# B&R Automation Studio project mvDemoTrak
Automation Studio 4.12.3.127 SP; technology packages: mapp 5.22.1, mappCockpit 5.22.0, mappMotion 5.22.1, mappView 5.22.1

## Configuration CP1685

CPU X20CP1685, AutomationRuntime D4.93, Build 6.3.0, Safety 0.0, Vc 

### Task classes (Cpu.sw)
```
Cyclic#1 (cycle 2000 us, tolerance 0 us):
  VisuTask <- VisuPackage.VisuTask.prg
Cyclic#2 (cycle 10000 us, tolerance 10000 us):
  AlarmXTask <- VisuPackage.AlarmXTask.prg
Binaries: FWRules, arsvcreg, TCData, TCLang, udbdef, mvLoader, CfgAlList, iomap, TC, Role, arconfig, asfw, ashwac, sysconf, CfgAlHist, User, ashwd
Libraries: standard, MpAlarmX, MpBase, astime, runtime, MpServer, AsBrStr, sys_lib, asieccon, arssl, dataobj, aruser, McBase, CoTrace, AsZip, FileIO
```

### Hardware
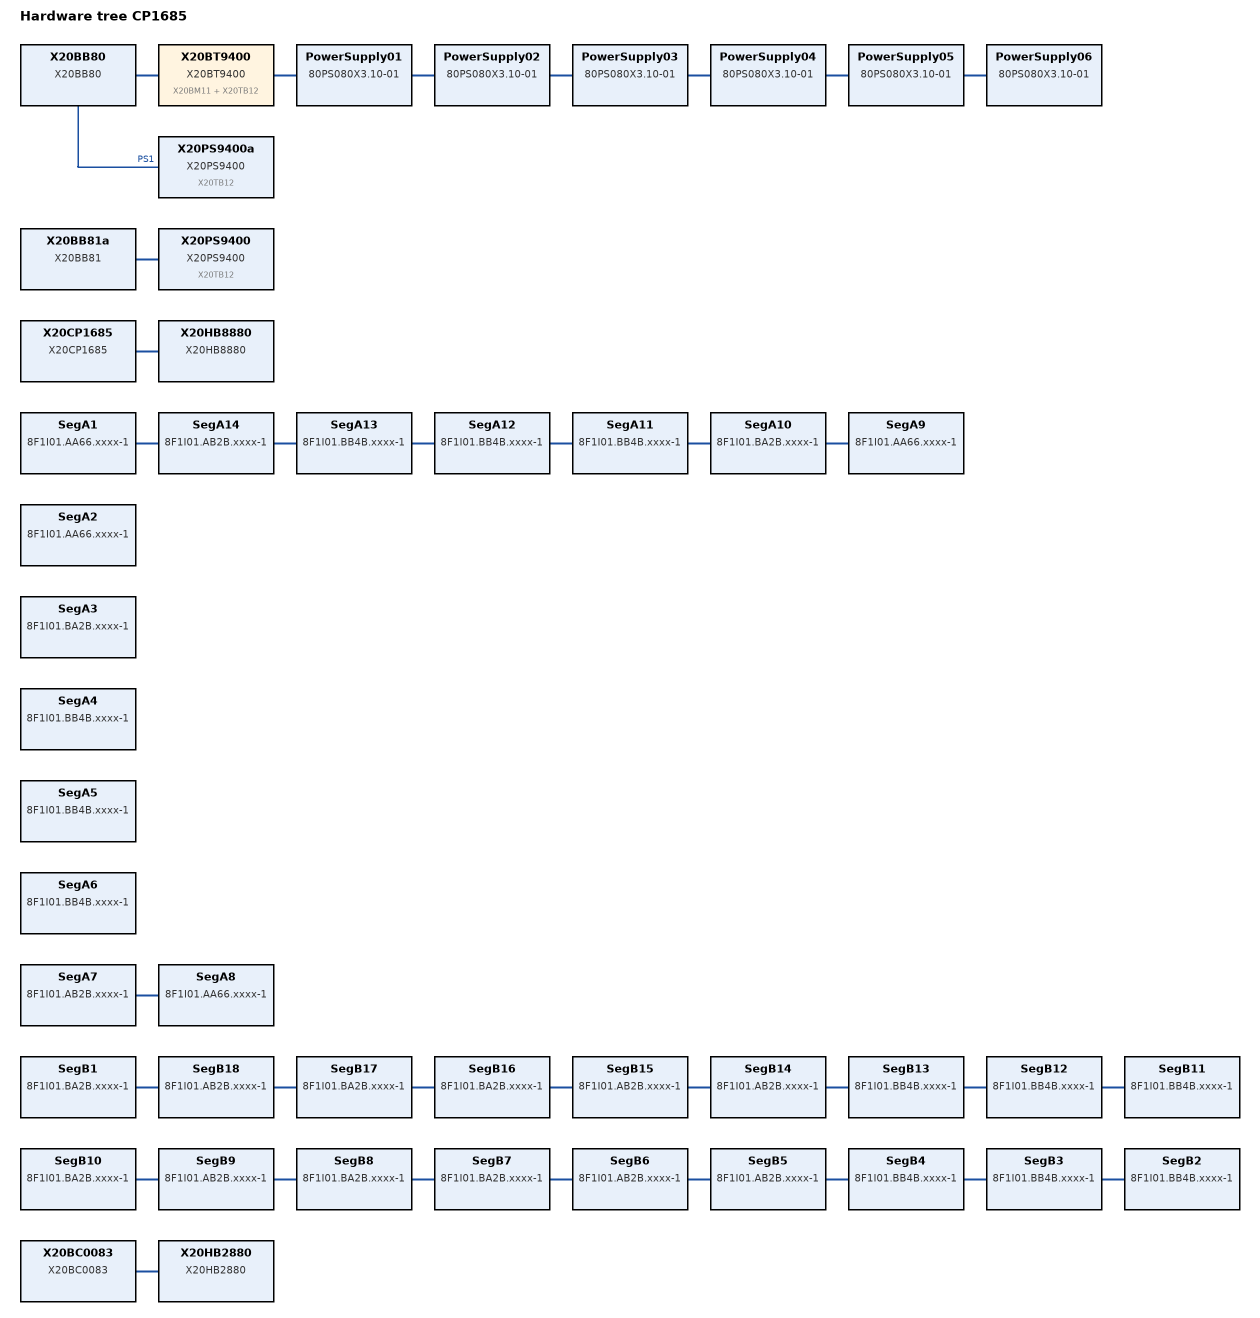
```
PowerSupply01 : 80PS080X3.10-01 v1.5.0.0  [X2X1 -> X20BT9400.X2X1 [Cable Type=X2XCable, Length=10, Version=1.0.0.3]]
  Supervision = off
PowerSupply02 : 80PS080X3.10-01 v1.5.0.0  [X2X1 -> PowerSupply01.X2X2 [Cable Type=X2XCable, Length=10, Version=1.0.0.3]]
  Supervision = off
PowerSupply03 : 80PS080X3.10-01 v1.5.0.0  [X2X1 -> PowerSupply02.X2X2 [Cable Type=X2XCable, Length=10, Version=1.0.0.3]]
  Supervision = off
PowerSupply04 : 80PS080X3.10-01 v1.5.0.0  [X2X1 -> PowerSupply03.X2X2 [Cable Type=X2XCable, Length=10, Version=1.0.0.3]]
  Supervision = off
PowerSupply05 : 80PS080X3.10-01 v1.5.0.0  [X2X1 -> PowerSupply04.X2X2 [Cable Type=X2XCable, Length=10, Version=1.0.0.3]]
  Supervision = off
PowerSupply06 : 80PS080X3.10-01 v1.5.0.0  [X2X1 -> PowerSupply05.X2X2 [Cable Type=X2XCable, Length=10, Version=1.0.0.3]]
  Supervision = off
SegA1 : 8F1I01.AA66.xxxx-1 v1.0.0.2  [PLK1 -> SegA2.PLK2 (NodeNumber=1) [Cable Type=PowerlinkCable, Length=10, Version=1.0.0.3]; PLK2 -> SegA14.PLK1 (NodeNumber=1) [Cable Type=PowerlinkCable, Length=10, Version=1.0.0.3]; PLK3 -> X20HB8880.ETH2 (NodeNumber=1) [Cable Type=PowerlinkCable, Length=10, Version=1.0.0.3]]
  DriveConfiguration:
    McTypeID = LLMConfig
  DriveConfiguration/Segment:
    Shape = STRAIGHT660
    SegmentReference = gSegA1
    SegmentSectorDirection = Positive
    ElongationCompensation = UseAssemblySetting
    StopReaction = UseAssemblySetting
    SpeedFilter = UseAssemblySetting
SegA10 : 8F1I01.BA2B.xxxx-1 v1.0.0.2  [PLK1 -> SegA11.PLK2 (NodeNumber=25) [Cable Type=PowerlinkCable, Length=10, Version=1.0.0.3]; PLK2 -> SegA9.PLK1 (NodeNumber=25) [Cable Type=PowerlinkCable, Length=10, Version=1.0.0.3]]
  DriveConfiguration:
    McTypeID = LLMConfig
  DriveConfiguration/Segment:
    Shape = CIRCULAR_TO_STRAIGHT105
    SegmentReference = gSegA10
    SegmentSectorDirection = Positive
    ElongationCompensation = UseAssemblySetting
    StopReaction = UseAssemblySetting
    SpeedFilter = UseAssemblySetting
SegA11 : 8F1I01.BB4B.xxxx-1 v1.0.0.2  [PLK1 -> SegA12.PLK2 (NodeNumber=24) [Cable Type=PowerlinkCable, Length=10, Version=1.0.0.3]; PLK2 -> SegA10.PLK1 (NodeNumber=24) [Cable Type=PowerlinkCable, Length=10, Version=1.0.0.3]]
  DriveConfiguration:
    McTypeID = LLMConfig
  DriveConfiguration/Segment:
    Shape = CIRCULAR
    SegmentReference = gSegA11
    SegmentSectorDirection = Positive
    ElongationCompensation = UseAssemblySetting
    StopReaction = UseAssemblySetting
    SpeedFilter = UseAssemblySetting
SegA12 : 8F1I01.BB4B.xxxx-1 v1.0.0.2  [PLK1 -> SegA13.PLK2 (NodeNumber=23) [Cable Type=PowerlinkCable, Length=10, Version=1.0.0.3]; PLK2 -> SegA11.PLK1 (NodeNumber=23) [Cable Type=PowerlinkCable, Length=10, Version=1.0.0.3]]
  DriveConfiguration:
    McTypeID = LLMConfig
  DriveConfiguration/Segment:
    Shape = CIRCULAR
    SegmentReference = gSegA12
    SegmentSectorDirection = Positive
    ElongationCompensation = UseAssemblySetting
    StopReaction = UseAssemblySetting
    SpeedFilter = UseAssemblySetting
SegA13 : 8F1I01.BB4B.xxxx-1 v1.0.0.2  [PLK1 -> SegA14.PLK2 (NodeNumber=22) [Cable Type=PowerlinkCable, Length=10, Version=1.0.0.3]; PLK2 -> SegA12.PLK1 (NodeNumber=22) [Cable Type=PowerlinkCable, Length=10, Version=1.0.0.3]]
  DriveConfiguration:
    McTypeID = LLMConfig
  DriveConfiguration/Segment:
    Shape = CIRCULAR
    SegmentReference = gSegA13
    SegmentSectorDirection = Positive
    ElongationCompensation = UseAssemblySetting
    StopReaction = UseAssemblySetting
    SpeedFilter = UseAssemblySetting
SegA14 : 8F1I01.AB2B.xxxx-1 v1.0.0.2  [PLK1 -> SegA1.PLK2 (NodeNumber=21) [Cable Type=PowerlinkCable, Length=10, Version=1.0.0.3]; PLK2 -> SegA13.PLK1 (NodeNumber=21) [Cable Type=PowerlinkCable, Length=10, Version=1.0.0.3]]
  DriveConfiguration:
    McTypeID = LLMConfig
  DriveConfiguration/Segment:
    Shape = STRAIGHT105_TO_CIRCULAR
    SegmentReference = gSegA14
    SegmentSectorDirection = Positive
    ElongationCompensation = UseAssemblySetting
    StopReaction = UseAssemblySetting
    SpeedFilter = UseAssemblySetting
SegA2 : 8F1I01.AA66.xxxx-1 v1.0.0.2  [PLK1 -> SegA3.PLK2 (NodeNumber=2) [Cable Type=PowerlinkCable, Length=10, Version=1.0.0.3]; PLK2 -> SegA1.PLK1 (NodeNumber=2) [Cable Type=PowerlinkCable, Length=10, Version=1.0.0.3]]
  DriveConfiguration:
    McTypeID = LLMConfig
  DriveConfiguration/Segment:
    Shape = STRAIGHT660
    SegmentReference = gSegA2
    SegmentSectorDirection = Positive
    ElongationCompensation = UseAssemblySetting
    StopReaction = UseAssemblySetting
    SpeedFilter = UseAssemblySetting
SegA3 : 8F1I01.BA2B.xxxx-1 v1.0.0.2  [PLK1 -> SegA4.PLK2 (NodeNumber=27) [Cable Type=PowerlinkCable, Length=10, Version=1.0.0.3]; PLK2 -> SegA2.PLK1 (NodeNumber=27) [Cable Type=PowerlinkCable, Length=10, Version=1.0.0.3]]
  DriveConfiguration:
    McTypeID = LLMConfig
  DriveConfiguration/Segment:
    Shape = CIRCULAR_TO_STRAIGHT105
    SegmentReference = gSegA3
    SegmentSectorDirection = Positive
    ElongationCompensation = UseAssemblySetting
    StopReaction = UseAssemblySetting
    SpeedFilter = UseAssemblySetting
SegA4 : 8F1I01.BB4B.xxxx-1 v1.0.0.2  [PLK1 -> SegA5.PLK2 (NodeNumber=28) [Cable Type=PowerlinkCable, Length=10, Version=1.0.0.3]; PLK2 -> SegA3.PLK1 (NodeNumber=28) [Cable Type=PowerlinkCable, Length=10, Version=1.0.0.3]]
  DriveConfiguration:
    McTypeID = LLMConfig
  DriveConfiguration/Segment:
    Shape = CIRCULAR
    SegmentReference = gSegA4
    SegmentSectorDirection = Positive
    ElongationCompensation = UseAssemblySetting
    StopReaction = UseAssemblySetting
    SpeedFilter = UseAssemblySetting
SegA5 : 8F1I01.BB4B.xxxx-1 v1.0.0.2  [PLK1 -> SegA6.PLK2 (NodeNumber=29) [Cable Type=PowerlinkCable, Length=10, Version=1.0.0.3]; PLK2 -> SegA4.PLK1 (NodeNumber=29) [Cable Type=PowerlinkCable, Length=10, Version=1.0.0.3]]
  DriveConfiguration:
    McTypeID = LLMConfig
  DriveConfiguration/Segment:
    Shape = CIRCULAR
    SegmentReference = gSegA5
    SegmentSectorDirection = Positive
    ElongationCompensation = UseAssemblySetting
    StopReaction = UseAssemblySetting
    SpeedFilter = UseAssemblySetting
SegA6 : 8F1I01.BB4B.xxxx-1 v1.0.0.2  [PLK1 -> SegA7.PLK2 (NodeNumber=30) [Cable Type=PowerlinkCable, Length=10, Version=1.0.0.3]; PLK2 -> SegA5.PLK1 (NodeNumber=30) [Cable Type=PowerlinkCable, Length=10, Version=1.0.0.3]]
  DriveConfiguration:
    McTypeID = LLMConfig
  DriveConfiguration/Segment:
    Shape = CIRCULAR
    SegmentReference = gSegA6
    SegmentSectorDirection = Positive
    ElongationCompensation = UseAssemblySetting
    StopReaction = UseAssemblySetting
    SpeedFilter = UseAssemblySetting
SegA7 : 8F1I01.AB2B.xxxx-1 v1.0.0.2  [PLK1 -> SegA8.PLK2 (NodeNumber=31) [Cable Type=PowerlinkCable, Length=10, Version=1.0.0.3]; PLK2 -> SegA6.PLK1 (NodeNumber=31) [Cable Type=PowerlinkCable, Length=10, Version=1.0.0.3]]
  DriveConfiguration:
    McTypeID = LLMConfig
  DriveConfiguration/Segment:
    Shape = STRAIGHT105_TO_CIRCULAR
    SegmentReference = gSegA7
    SegmentSectorDirection = Positive
    ElongationCompensation = UseAssemblySetting
    StopReaction = UseAssemblySetting
    SpeedFilter = UseAssemblySetting
SegA8 : 8F1I01.AA66.xxxx-1 v1.0.0.2  [PLK2 -> SegA7.PLK1 (NodeNumber=32) [Cable Type=PowerlinkCable, Length=10, Version=1.0.0.3]]
  DriveConfiguration:
    McTypeID = LLMConfig
  DriveConfiguration/Segment:
    Shape = STRAIGHT660
    SegmentReference = gSegA8
    SegmentSectorDirection = Positive
    ElongationCompensation = UseAssemblySetting
    StopReaction = UseAssemblySetting
    SpeedFilter = UseAssemblySetting
SegA9 : 8F1I01.AA66.xxxx-1 v1.0.0.2  [PLK1 -> SegA10.PLK2 (NodeNumber=26) [Cable Type=PowerlinkCable, Length=10, Version=1.0.0.3]]
  DriveConfiguration:
    McTypeID = LLMConfig
  DriveConfiguration/Segment:
    Shape = STRAIGHT660
    SegmentReference = gSegA9
    SegmentSectorDirection = Positive
    ElongationCompensation = UseAssemblySetting
    StopReaction = UseAssemblySetting
    SpeedFilter = UseAssemblySetting
SegB1 : 8F1I01.BA2B.xxxx-1 v1.0.0.2  [PLK1 -> SegB2.PLK2 (NodeNumber=3) [Cable Type=PowerlinkCable, Length=10, Version=1.0.0.3]; PLK2 -> SegB18.PLK1 (NodeNumber=3) [Cable Type=PowerlinkCable, Length=10, Version=1.0.0.3]; PLK3 -> X20HB2880.ETH2 (NodeNumber=3) [Cable Type=PowerlinkCable, Length=10, Version=1.0.0.3]]
  DriveConfiguration:
    McTypeID = LLMConfig
  DriveConfiguration/Segment:
    Shape = CIRCULAR_TO_STRAIGHT105
    SegmentReference = gSegB1
    SegmentSectorDirection = Positive
    ElongationCompensation = UseAssemblySetting
    StopReaction = UseAssemblySetting
    SpeedFilter = UseAssemblySetting
SegB10 : 8F1I01.BA2B.xxxx-1 v1.0.0.2  [PLK2 -> SegB9.PLK1 (NodeNumber=12) [Cable Type=PowerlinkCable, Length=10, Version=1.0.0.3]]
  DriveConfiguration:
    McTypeID = LLMConfig
  DriveConfiguration/Segment:
    Shape = CIRCULAR_TO_STRAIGHT105
    SegmentReference = gSegB10
    SegmentSectorDirection = Positive
    ElongationCompensation = UseAssemblySetting
    StopReaction = UseAssemblySetting
    SpeedFilter = UseAssemblySetting
SegB11 : 8F1I01.BB4B.xxxx-1 v1.0.0.2  [PLK1 -> SegB12.PLK2 (NodeNumber=11) [Cable Type=PowerlinkCable, Length=10, Version=1.0.0.3]]
  DriveConfiguration:
    McTypeID = LLMConfig
  DriveConfiguration/Segment:
    Shape = CIRCULAR
    SegmentReference = gSegB11
    SegmentSectorDirection = Positive
    ElongationCompensation = UseAssemblySetting
    StopReaction = UseAssemblySetting
    SpeedFilter = UseAssemblySetting
SegB12 : 8F1I01.BB4B.xxxx-1 v1.0.0.2  [PLK1 -> SegB13.PLK2 (NodeNumber=10) [Cable Type=PowerlinkCable, Length=10, Version=1.0.0.3]; PLK2 -> SegB11.PLK1 (NodeNumber=10) [Cable Type=PowerlinkCable, Length=10, Version=1.0.0.3]]
  DriveConfiguration:
    McTypeID = LLMConfig
  DriveConfiguration/Segment:
    Shape = CIRCULAR
    SegmentReference = gSegB12
    SegmentSectorDirection = Positive
    ElongationCompensation = UseAssemblySetting
    StopReaction = UseAssemblySetting
    SpeedFilter = UseAssemblySetting
SegB13 : 8F1I01.BB4B.xxxx-1 v1.0.0.2  [PLK1 -> SegB14.PLK2 (NodeNumber=9) [Cable Type=PowerlinkCable, Length=10, Version=1.0.0.3]; PLK2 -> SegB12.PLK1 (NodeNumber=9) [Cable Type=PowerlinkCable, Length=10, Version=1.0.0.3]]
  DriveConfiguration:
    McTypeID = LLMConfig
  DriveConfiguration/Segment:
    Shape = CIRCULAR
    SegmentReference = gSegB13
    SegmentSectorDirection = Positive
    ElongationCompensation = UseAssemblySetting
    StopReaction = UseAssemblySetting
    SpeedFilter = UseAssemblySetting
SegB14 : 8F1I01.AB2B.xxxx-1 v1.0.0.2  [PLK1 -> SegB15.PLK2 (NodeNumber=8) [Cable Type=PowerlinkCable, Length=10, Version=1.0.0.3]; PLK2 -> SegB13.PLK1 (NodeNumber=8) [Cable Type=PowerlinkCable, Length=10, Version=1.0.0.3]]
  DriveConfiguration:
    McTypeID = LLMConfig
  DriveConfiguration/Segment:
    Shape = STRAIGHT105_TO_CIRCULAR
    SegmentReference = gSegB14
    SegmentSectorDirection = Positive
    ElongationCompensation = UseAssemblySetting
    StopReaction = UseAssemblySetting
    SpeedFilter = UseAssemblySetting
SegB15 : 8F1I01.AB2B.xxxx-1 v1.0.0.2  [PLK1 -> SegB16.PLK2 (NodeNumber=7) [Cable Type=PowerlinkCable, Length=10, Version=1.0.0.3]; PLK2 -> SegB14.PLK1 (NodeNumber=7) [Cable Type=PowerlinkCable, Length=10, Version=1.0.0.3]]
  DriveConfiguration:
    McTypeID = LLMConfig
  DriveConfiguration/Segment:
    Shape = STRAIGHT105_TO_CIRCULAR
    SegmentReference = gSegB15
    SegmentSectorDirection = Positive
    ElongationCompensation = UseAssemblySetting
    StopReaction = UseAssemblySetting
    SpeedFilter = UseAssemblySetting
SegB16 : 8F1I01.BA2B.xxxx-1 v1.0.0.2  [PLK1 -> SegB17.PLK2 (NodeNumber=6) [Cable Type=PowerlinkCable, Length=10, Version=1.0.0.3]; PLK2 -> SegB15.PLK1 (NodeNumber=6) [Cable Type=PowerlinkCable, Length=10, Version=1.0.0.3]]
  DriveConfiguration:
    McTypeID = LLMConfig
  DriveConfiguration/Segment:
    Shape = CIRCULAR_TO_STRAIGHT105
    SegmentReference = gSegB16
    SegmentSectorDirection = Positive
    ElongationCompensation = UseAssemblySetting
    StopReaction = UseAssemblySetting
    SpeedFilter = UseAssemblySetting
SegB17 : 8F1I01.BA2B.xxxx-1 v1.0.0.2  [PLK1 -> SegB18.PLK2 (NodeNumber=5) [Cable Type=PowerlinkCable, Length=10, Version=1.0.0.3]; PLK2 -> SegB16.PLK1 (NodeNumber=5) [Cable Type=PowerlinkCable, Length=10, Version=1.0.0.3]]
  DriveConfiguration:
    McTypeID = LLMConfig
  DriveConfiguration/Segment:
    Shape = CIRCULAR_TO_STRAIGHT105
    SegmentReference = gSegB17
    SegmentSectorDirection = Positive
    ElongationCompensation = UseAssemblySetting
    StopReaction = UseAssemblySetting
    SpeedFilter = UseAssemblySetting
SegB18 : 8F1I01.AB2B.xxxx-1 v1.0.0.2  [PLK1 -> SegB1.PLK2 (NodeNumber=4) [Cable Type=PowerlinkCable, Length=10, Version=1.0.0.3]; PLK2 -> SegB17.PLK1 (NodeNumber=4) [Cable Type=PowerlinkCable, Length=10, Version=1.0.0.3]]
  DriveConfiguration:
    McTypeID = LLMConfig
  DriveConfiguration/Segment:
    Shape = STRAIGHT105_TO_CIRCULAR
    SegmentReference = gSegB18
    SegmentSectorDirection = Positive
    ElongationCompensation = UseAssemblySetting
    StopReaction = UseAssemblySetting
    SpeedFilter = UseAssemblySetting
SegB2 : 8F1I01.BB4B.xxxx-1 v1.0.0.2  [PLK1 -> SegB3.PLK2 (NodeNumber=13) [Cable Type=PowerlinkCable, Length=10, Version=1.0.0.3]; PLK2 -> SegB1.PLK1 (NodeNumber=13) [Cable Type=PowerlinkCable, Length=10, Version=1.0.0.3]]
  DriveConfiguration:
    McTypeID = LLMConfig
  DriveConfiguration/Segment:
    Shape = CIRCULAR
    SegmentReference = gSegB2
    SegmentSectorDirection = Positive
    ElongationCompensation = UseAssemblySetting
    StopReaction = UseAssemblySetting
    SpeedFilter = UseAssemblySetting
SegB3 : 8F1I01.BB4B.xxxx-1 v1.0.0.2  [PLK1 -> SegB4.PLK2 (NodeNumber=14) [Cable Type=PowerlinkCable, Length=10, Version=1.0.0.3]; PLK2 -> SegB2.PLK1 (NodeNumber=14) [Cable Type=PowerlinkCable, Length=10, Version=1.0.0.3]]
  DriveConfiguration:
    McTypeID = LLMConfig
  DriveConfiguration/Segment:
    Shape = CIRCULAR
    SegmentReference = gSegB3
    SegmentSectorDirection = Positive
    ElongationCompensation = UseAssemblySetting
    StopReaction = UseAssemblySetting
    SpeedFilter = UseAssemblySetting
SegB4 : 8F1I01.BB4B.xxxx-1 v1.0.0.2  [PLK1 -> SegB5.PLK2 (NodeNumber=15) [Cable Type=PowerlinkCable, Length=10, Version=1.0.0.3]; PLK2 -> SegB3.PLK1 (NodeNumber=15) [Cable Type=PowerlinkCable, Length=10, Version=1.0.0.3]]
  DriveConfiguration:
    McTypeID = LLMConfig
  DriveConfiguration/Segment:
    Shape = CIRCULAR
    SegmentReference = gSegB4
    SegmentSectorDirection = Positive
    ElongationCompensation = UseAssemblySetting
    StopReaction = UseAssemblySetting
    SpeedFilter = UseAssemblySetting
SegB5 : 8F1I01.AB2B.xxxx-1 v1.0.0.2  [PLK1 -> SegB6.PLK2 (NodeNumber=16) [Cable Type=PowerlinkCable, Length=10, Version=1.0.0.3]; PLK2 -> SegB4.PLK1 (NodeNumber=16) [Cable Type=PowerlinkCable, Length=10, Version=1.0.0.3]]
  DriveConfiguration:
    McTypeID = LLMConfig
  DriveConfiguration/Segment:
    Shape = STRAIGHT105_TO_CIRCULAR
    SegmentReference = gSegB5
    SegmentSectorDirection = Positive
    ElongationCompensation = UseAssemblySetting
    StopReaction = UseAssemblySetting
    SpeedFilter = UseAssemblySetting
SegB6 : 8F1I01.AB2B.xxxx-1 v1.0.0.2  [PLK1 -> SegB7.PLK2 (NodeNumber=17) [Cable Type=PowerlinkCable, Length=10, Version=1.0.0.3]; PLK2 -> SegB5.PLK1 (NodeNumber=17) [Cable Type=PowerlinkCable, Length=10, Version=1.0.0.3]]
  DriveConfiguration:
    McTypeID = LLMConfig
  DriveConfiguration/Segment:
    Shape = STRAIGHT105_TO_CIRCULAR
    SegmentReference = gSegB6
    SegmentSectorDirection = Positive
    ElongationCompensation = UseAssemblySetting
    StopReaction = UseAssemblySetting
    SpeedFilter = UseAssemblySetting
SegB7 : 8F1I01.BA2B.xxxx-1 v1.0.0.2  [PLK1 -> SegB8.PLK2 (NodeNumber=18) [Cable Type=PowerlinkCable, Length=10, Version=1.0.0.3]; PLK2 -> SegB6.PLK1 (NodeNumber=18) [Cable Type=PowerlinkCable, Length=10, Version=1.0.0.3]]
  DriveConfiguration:
    McTypeID = LLMConfig
  DriveConfiguration/Segment:
    Shape = CIRCULAR_TO_STRAIGHT105
    SegmentReference = gSegB7
    SegmentSectorDirection = Positive
    ElongationCompensation = UseAssemblySetting
    StopReaction = UseAssemblySetting
    SpeedFilter = UseAssemblySetting
SegB8 : 8F1I01.BA2B.xxxx-1 v1.0.0.2  [PLK1 -> SegB9.PLK2 (NodeNumber=20) [Cable Type=PowerlinkCable, Length=10, Version=1.0.0.3]; PLK2 -> SegB7.PLK1 (NodeNumber=20) [Cable Type=PowerlinkCable, Length=10, Version=1.0.0.3]]
  DriveConfiguration:
    McTypeID = LLMConfig
  DriveConfiguration/Segment:
    Shape = CIRCULAR_TO_STRAIGHT105
    SegmentReference = gSegB8
    SegmentSectorDirection = Positive
    ElongationCompensation = UseAssemblySetting
    StopReaction = UseAssemblySetting
    SpeedFilter = UseAssemblySetting
SegB9 : 8F1I01.AB2B.xxxx-1 v1.0.0.2  [PLK1 -> SegB10.PLK2 (NodeNumber=19) [Cable Type=PowerlinkCable, Length=10, Version=1.0.0.3]; PLK2 -> SegB8.PLK1 (NodeNumber=19) [Cable Type=PowerlinkCable, Length=10, Version=1.0.0.3]]
  DriveConfiguration:
    McTypeID = LLMConfig
  DriveConfiguration/Segment:
    Shape = STRAIGHT105_TO_CIRCULAR
    SegmentReference = gSegB9
    SegmentSectorDirection = Positive
    ElongationCompensation = UseAssemblySetting
    StopReaction = UseAssemblySetting
    SpeedFilter = UseAssemblySetting
X20BB80 : X20BB80 v1.1.0.0
X20BB81a : X20BB81 v1.1.0.0
  Connector IF1:
    ActivateX2X = 0
X20BC0083 : X20BC0083 v2.14.0.0  [PLK1 -> X20HB2880.ETH1 (NodeNumber=33) [Cable Type=PowerlinkCable, Length=10, Version=1.0.0.3]; SL -> X20BB80.SL1]
  Supervision = off
X20BM11 : X20BM11 v1.1.0.0  [X2X1 -> X20BB80.IF1]
X20BT9400 : X20BT9400 v1.3.0.0  [SS1 -> X20TB12b.SS; SL -> X20BM11.SL1]
  Supervision = off
X20CP1685 : X20CP1685 v1.7.2.0
  Connector IF2:
    ActivateDevice = 1
    Mode = Manual
    InternetAddress = 192.168.0.105  // //10.49.40.211
    SubnetMask = 255.255.255.0
    ActivateSnmp = 2
  ConfigurationID = mvDemoTrak_CP1685
  MotionLoggerSize = 2048000
  EnableUsbRemoteInstall = 1
  TimerDeviceType = EPLX2X
  TimerDevice = X20CP1685.IF3
  TaskClassIdleTime = 2000
  Cyclic1Duration = 2000
  Cyclic1Tolerance = 0
  Cyclic2Duration = 10000
  Cyclic2Tolerance = 10000
  FileDevice1
  FileDeviceName1 = SvgData
  FileDevicePath1 = F:\web\SvgData
  FileDevice2
  FileDeviceName2 = Diagnosis
  FileDevicePath2 = F:\web\Diagnosis
  FtpUser1
  FtpUsername1 = Admin
  FtpUserPassword1 = b2dkeklN0DR4HlzomfG8N5dlVtI3Hrgd5HBjTL6T4A4=  // pw: admin
  FtpUserSalt1 = LZ6GLOae
  FTPAccessRight1 = 0
  FTPdevice1 = ALL
  WebServerWebDir = F:\web  // default: web\
  ActivateOpcUa = 1
  OpcUaInformationModels_PV_Version = 1
X20HB2880 : X20HB2880 v1.2.0.0  [ETH1 -> X20BC0083.PLK1 [Cable Type=PowerlinkCable, Length=10, Version=1.0.0.3]; ETH2 -> SegB1.PLK3 [Cable Type=PowerlinkCable, Length=10, Version=1.0.0.3]; SS -> X20BB81a.SS1]
X20HB8880 : X20HB8880 v1.1.0.0  [ETH1 -> X20CP1685.IF3 [Cable Type=PowerlinkCable, Length=10, Version=1.0.0.3]; ETH2 -> SegA1.PLK3 [Cable Type=PowerlinkCable, Length=10, Version=1.0.0.3]; SL -> X20BB81a.SL1]
X20PS9400 : X20PS9400 v1.8.0.0  [SS1 -> X20TB12.SS; PS -> X20BB81a.PS1]
  Supervision = off
X20PS9400a : X20PS9400 v1.8.0.0  [SS1 -> X20TB12a.SS; PS -> X20BB80.PS1]
  Supervision = off
X20TB12 : X20TB12 v1.0.0.0
X20TB12a : X20TB12 v1.0.0.0
X20TB12b : X20TB12 v1.0.0.0
```

### CfgAlList.mpalarmxcore - X20CP1685/mappServices/CfgAlList.mpalarmxcore
```
Element gAlarmXCore (Type=mpalarmxcore)
  mapp.AlarmX.Core:
    BySeverity:
      [0]:
        Severity = 10
        [0] = Reaction
          Name = ActWarning
      [1]:
        Severity = 50
        [0] = Reaction
          Name = ActErrorMed
      [2]:
        Severity = 100
        [0] = Reaction
          Name = ActError
  mapp.AlarmX.Core.Configuration:
    [0]:
      Name = AL_AlarmMeldung
      Message = AlarmMeldung
      Code = 100
      Severity = 100
      Behavior = DiscreteValueMonitoring
        Monitoring:
          MonitoredPV = ::AlarmXTask:tmpErrorID
          TriggerValues:
            [0] = 100
    [1]:
      Name = AL_AlarmMeldung1
      Message = AlarmMeldung
      Code = 101
      Severity = 100
      Behavior = DiscreteValueMonitoring
        Monitoring:
          MonitoredPV = ::AlarmXTask:tmpErrorID
          TriggerValues:
            [0] = 101
    [2]:
      Name = AL_AlarmMedMeldung
      Message = AlarmMedMeldung
      Code = 50
      Severity = 50
      Behavior = DiscreteValueMonitoring
        Monitoring:
          MonitoredPV = ::AlarmXTask:tmpErrorID
          TriggerValues:
            [0] = 50
    [3]:
      Name = AL_AlarmMedMeldung1
      Message = AlarmMedMeldung1
      Code = 51
      Severity = 50
      Behavior = DiscreteValueMonitoring
        Monitoring:
          MonitoredPV = ::AlarmXTask:tmpErrorID
          TriggerValues:
            [0] = 51
    [4]:
      Name = AL_Warnung
      Message = Warnung
      Code = 10
      Severity = 10
      Behavior = DiscreteValueMonitoring
        Monitoring:
          MonitoredPV = ::AlarmXTask:tmpErrorID
          TriggerValues:
            [0] = 10
    [5]:
      Name = AL_Warnung1
      Message = Warnung1
      Code = 11
      Severity = 10
      Behavior = DiscreteValueMonitoring
        Monitoring:
          MonitoredPV = ::AlarmXTask:tmpErrorID
          TriggerValues:
            [0] = 11
  mapp.AlarmX.Core.Categories:
    [0]:
      Name = CatWarning
      SourceProperty:
        Severity = 10
    [1]:
      Name = CatErrorMed
      SourceProperty:
        Severity = 50
    [2]:
      Name = CatError
      SourceProperty:
        Severity = 100
```

## Configuration CP3686X

CPU X20CP3686X, AutomationRuntime D4.93, Build 6.3.0, Safety 0.0, Vc 

### Hardware
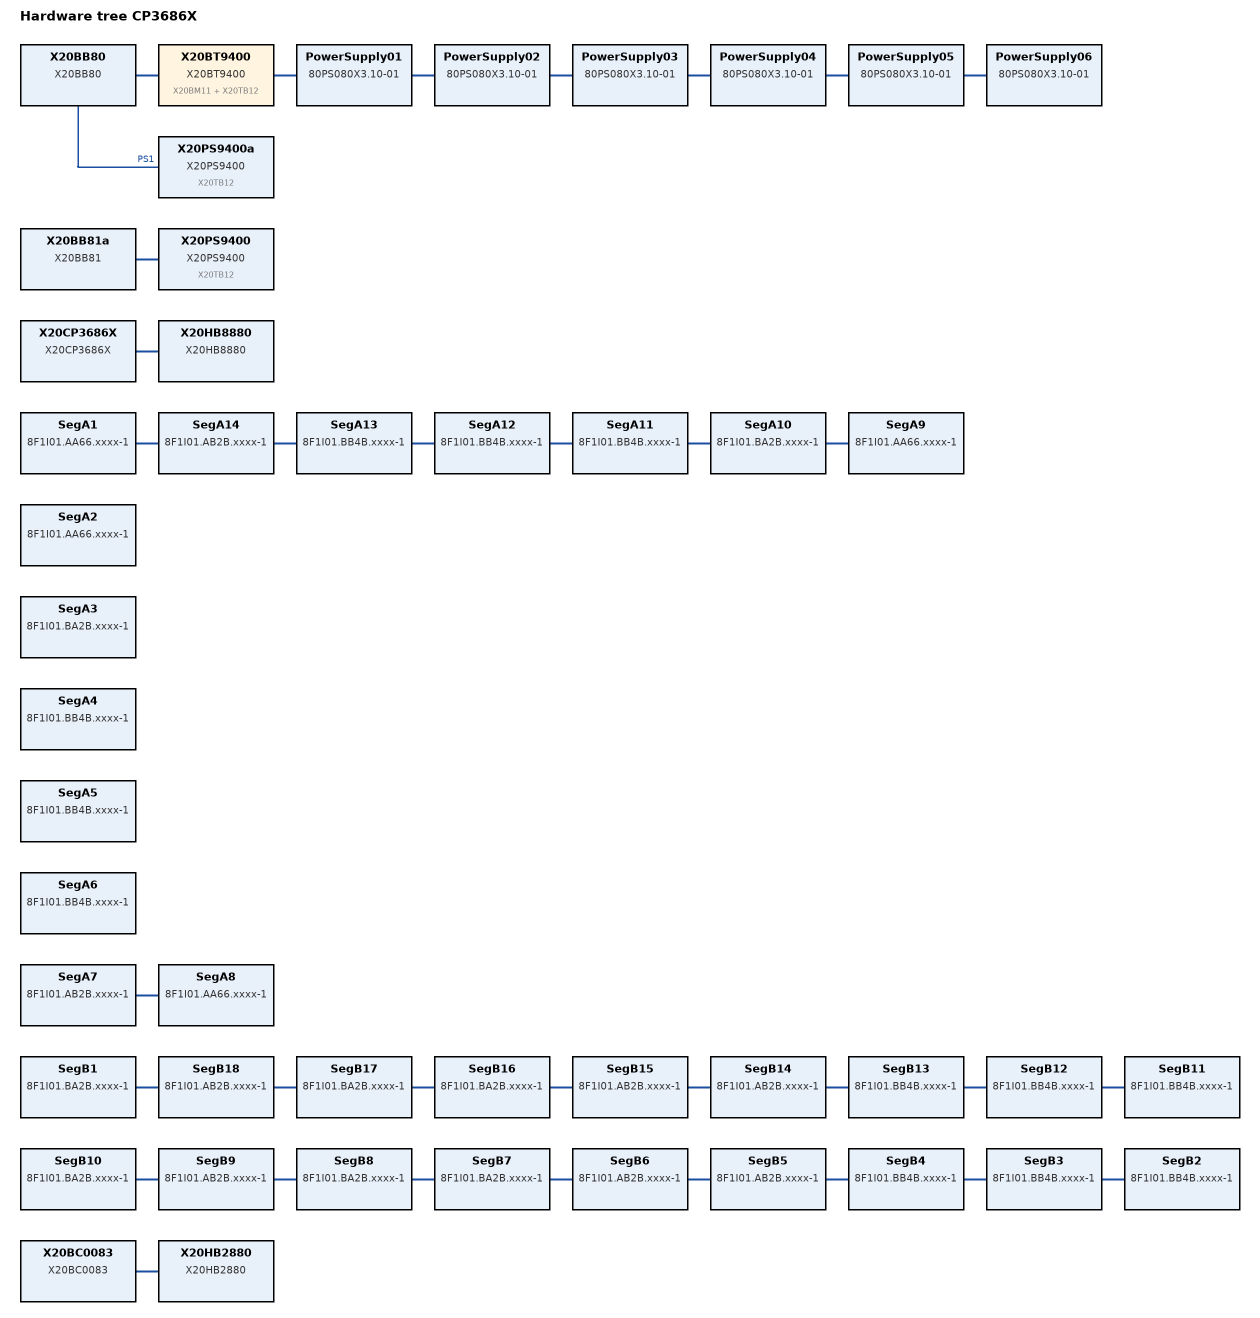
```
PowerSupply01 : 80PS080X3.10-01 v1.5.0.0  [X2X1 -> X20BT9400.X2X1 [Cable Type=X2XCable, Length=10, Version=1.0.0.3]]
  Supervision = off
PowerSupply02 : 80PS080X3.10-01 v1.5.0.0  [X2X1 -> PowerSupply01.X2X2 [Cable Type=X2XCable, Length=10, Version=1.0.0.3]]
  Supervision = off
PowerSupply03 : 80PS080X3.10-01 v1.5.0.0  [X2X1 -> PowerSupply02.X2X2 [Cable Type=X2XCable, Length=10, Version=1.0.0.3]]
  Supervision = off
PowerSupply04 : 80PS080X3.10-01 v1.5.0.0  [X2X1 -> PowerSupply03.X2X2 [Cable Type=X2XCable, Length=10, Version=1.0.0.3]]
  Supervision = off
PowerSupply05 : 80PS080X3.10-01 v1.5.0.0  [X2X1 -> PowerSupply04.X2X2 [Cable Type=X2XCable, Length=10, Version=1.0.0.3]]
  Supervision = off
PowerSupply06 : 80PS080X3.10-01 v1.5.0.0  [X2X1 -> PowerSupply05.X2X2 [Cable Type=X2XCable, Length=10, Version=1.0.0.3]]
  Supervision = off
SegA1 : 8F1I01.AA66.xxxx-1 v1.0.0.2  [PLK1 -> SegA2.PLK2 (NodeNumber=1) [Cable Type=PowerlinkCable, Length=10, Version=1.0.0.3]; PLK2 -> SegA14.PLK1 (NodeNumber=1) [Cable Type=PowerlinkCable, Length=10, Version=1.0.0.3]; PLK3 -> X20HB8880.ETH2 (NodeNumber=1) [Cable Type=PowerlinkCable, Length=10, Version=1.0.0.3]]
  DriveConfiguration:
    McTypeID = LLMConfig
  DriveConfiguration/Segment:
    Shape = STRAIGHT660
    SegmentReference = gSegA1
    SegmentSectorDirection = Positive
    ElongationCompensation = UseAssemblySetting
    StopReaction = UseAssemblySetting
    SpeedFilter = UseAssemblySetting
SegA10 : 8F1I01.BA2B.xxxx-1 v1.0.0.2  [PLK1 -> SegA11.PLK2 (NodeNumber=25) [Cable Type=PowerlinkCable, Length=10, Version=1.0.0.3]; PLK2 -> SegA9.PLK1 (NodeNumber=25) [Cable Type=PowerlinkCable, Length=10, Version=1.0.0.3]]
  DriveConfiguration:
    McTypeID = LLMConfig
  DriveConfiguration/Segment:
    Shape = CIRCULAR_TO_STRAIGHT105
    SegmentReference = gSegA10
    SegmentSectorDirection = Positive
    ElongationCompensation = UseAssemblySetting
    StopReaction = UseAssemblySetting
    SpeedFilter = UseAssemblySetting
SegA11 : 8F1I01.BB4B.xxxx-1 v1.0.0.2  [PLK1 -> SegA12.PLK2 (NodeNumber=24) [Cable Type=PowerlinkCable, Length=10, Version=1.0.0.3]; PLK2 -> SegA10.PLK1 (NodeNumber=24) [Cable Type=PowerlinkCable, Length=10, Version=1.0.0.3]]
  DriveConfiguration:
    McTypeID = LLMConfig
  DriveConfiguration/Segment:
    Shape = CIRCULAR
    SegmentReference = gSegA11
    SegmentSectorDirection = Positive
    ElongationCompensation = UseAssemblySetting
    StopReaction = UseAssemblySetting
    SpeedFilter = UseAssemblySetting
SegA12 : 8F1I01.BB4B.xxxx-1 v1.0.0.2  [PLK1 -> SegA13.PLK2 (NodeNumber=23) [Cable Type=PowerlinkCable, Length=10, Version=1.0.0.3]; PLK2 -> SegA11.PLK1 (NodeNumber=23) [Cable Type=PowerlinkCable, Length=10, Version=1.0.0.3]]
  DriveConfiguration:
    McTypeID = LLMConfig
  DriveConfiguration/Segment:
    Shape = CIRCULAR
    SegmentReference = gSegA12
    SegmentSectorDirection = Positive
    ElongationCompensation = UseAssemblySetting
    StopReaction = UseAssemblySetting
    SpeedFilter = UseAssemblySetting
SegA13 : 8F1I01.BB4B.xxxx-1 v1.0.0.2  [PLK1 -> SegA14.PLK2 (NodeNumber=22) [Cable Type=PowerlinkCable, Length=10, Version=1.0.0.3]; PLK2 -> SegA12.PLK1 (NodeNumber=22) [Cable Type=PowerlinkCable, Length=10, Version=1.0.0.3]]
  DriveConfiguration:
    McTypeID = LLMConfig
  DriveConfiguration/Segment:
    Shape = CIRCULAR
    SegmentReference = gSegA13
    SegmentSectorDirection = Positive
    ElongationCompensation = UseAssemblySetting
    StopReaction = UseAssemblySetting
    SpeedFilter = UseAssemblySetting
SegA14 : 8F1I01.AB2B.xxxx-1 v1.0.0.2  [PLK1 -> SegA1.PLK2 (NodeNumber=21) [Cable Type=PowerlinkCable, Length=10, Version=1.0.0.3]; PLK2 -> SegA13.PLK1 (NodeNumber=21) [Cable Type=PowerlinkCable, Length=10, Version=1.0.0.3]]
  DriveConfiguration:
    McTypeID = LLMConfig
  DriveConfiguration/Segment:
    Shape = STRAIGHT105_TO_CIRCULAR
    SegmentReference = gSegA14
    SegmentSectorDirection = Positive
    ElongationCompensation = UseAssemblySetting
    StopReaction = UseAssemblySetting
    SpeedFilter = UseAssemblySetting
SegA2 : 8F1I01.AA66.xxxx-1 v1.0.0.2  [PLK1 -> SegA3.PLK2 (NodeNumber=2) [Cable Type=PowerlinkCable, Length=10, Version=1.0.0.3]; PLK2 -> SegA1.PLK1 (NodeNumber=2) [Cable Type=PowerlinkCable, Length=10, Version=1.0.0.3]]
  DriveConfiguration:
    McTypeID = LLMConfig
  DriveConfiguration/Segment:
    Shape = STRAIGHT660
    SegmentReference = gSegA2
    SegmentSectorDirection = Positive
    ElongationCompensation = UseAssemblySetting
    StopReaction = UseAssemblySetting
    SpeedFilter = UseAssemblySetting
SegA3 : 8F1I01.BA2B.xxxx-1 v1.0.0.2  [PLK1 -> SegA4.PLK2 (NodeNumber=27) [Cable Type=PowerlinkCable, Length=10, Version=1.0.0.3]; PLK2 -> SegA2.PLK1 (NodeNumber=27) [Cable Type=PowerlinkCable, Length=10, Version=1.0.0.3]]
  DriveConfiguration:
    McTypeID = LLMConfig
  DriveConfiguration/Segment:
    Shape = CIRCULAR_TO_STRAIGHT105
    SegmentReference = gSegA3
    SegmentSectorDirection = Positive
    ElongationCompensation = UseAssemblySetting
    StopReaction = UseAssemblySetting
    SpeedFilter = UseAssemblySetting
SegA4 : 8F1I01.BB4B.xxxx-1 v1.0.0.2  [PLK1 -> SegA5.PLK2 (NodeNumber=28) [Cable Type=PowerlinkCable, Length=10, Version=1.0.0.3]; PLK2 -> SegA3.PLK1 (NodeNumber=28) [Cable Type=PowerlinkCable, Length=10, Version=1.0.0.3]]
  DriveConfiguration:
    McTypeID = LLMConfig
  DriveConfiguration/Segment:
    Shape = CIRCULAR
    SegmentReference = gSegA4
    SegmentSectorDirection = Positive
    ElongationCompensation = UseAssemblySetting
    StopReaction = UseAssemblySetting
    SpeedFilter = UseAssemblySetting
SegA5 : 8F1I01.BB4B.xxxx-1 v1.0.0.2  [PLK1 -> SegA6.PLK2 (NodeNumber=29) [Cable Type=PowerlinkCable, Length=10, Version=1.0.0.3]; PLK2 -> SegA4.PLK1 (NodeNumber=29) [Cable Type=PowerlinkCable, Length=10, Version=1.0.0.3]]
  DriveConfiguration:
    McTypeID = LLMConfig
  DriveConfiguration/Segment:
    Shape = CIRCULAR
    SegmentReference = gSegA5
    SegmentSectorDirection = Positive
    ElongationCompensation = UseAssemblySetting
    StopReaction = UseAssemblySetting
    SpeedFilter = UseAssemblySetting
SegA6 : 8F1I01.BB4B.xxxx-1 v1.0.0.2  [PLK1 -> SegA7.PLK2 (NodeNumber=30) [Cable Type=PowerlinkCable, Length=10, Version=1.0.0.3]; PLK2 -> SegA5.PLK1 (NodeNumber=30) [Cable Type=PowerlinkCable, Length=10, Version=1.0.0.3]]
  DriveConfiguration:
    McTypeID = LLMConfig
  DriveConfiguration/Segment:
    Shape = CIRCULAR
    SegmentReference = gSegA6
    SegmentSectorDirection = Positive
    ElongationCompensation = UseAssemblySetting
    StopReaction = UseAssemblySetting
    SpeedFilter = UseAssemblySetting
SegA7 : 8F1I01.AB2B.xxxx-1 v1.0.0.2  [PLK1 -> SegA8.PLK2 (NodeNumber=31) [Cable Type=PowerlinkCable, Length=10, Version=1.0.0.3]; PLK2 -> SegA6.PLK1 (NodeNumber=31) [Cable Type=PowerlinkCable, Length=10, Version=1.0.0.3]]
  DriveConfiguration:
    McTypeID = LLMConfig
  DriveConfiguration/Segment:
    Shape = STRAIGHT105_TO_CIRCULAR
    SegmentReference = gSegA7
    SegmentSectorDirection = Positive
    ElongationCompensation = UseAssemblySetting
    StopReaction = UseAssemblySetting
    SpeedFilter = UseAssemblySetting
SegA8 : 8F1I01.AA66.xxxx-1 v1.0.0.2  [PLK2 -> SegA7.PLK1 (NodeNumber=32) [Cable Type=PowerlinkCable, Length=10, Version=1.0.0.3]]
  DriveConfiguration:
    McTypeID = LLMConfig
  DriveConfiguration/Segment:
    Shape = STRAIGHT660
    SegmentReference = gSegA8
    SegmentSectorDirection = Positive
    ElongationCompensation = UseAssemblySetting
    StopReaction = UseAssemblySetting
    SpeedFilter = UseAssemblySetting
SegA9 : 8F1I01.AA66.xxxx-1 v1.0.0.2  [PLK1 -> SegA10.PLK2 (NodeNumber=26) [Cable Type=PowerlinkCable, Length=10, Version=1.0.0.3]]
  DriveConfiguration:
    McTypeID = LLMConfig
  DriveConfiguration/Segment:
    Shape = STRAIGHT660
    SegmentReference = gSegA9
    SegmentSectorDirection = Positive
    ElongationCompensation = UseAssemblySetting
    StopReaction = UseAssemblySetting
    SpeedFilter = UseAssemblySetting
SegB1 : 8F1I01.BA2B.xxxx-1 v1.0.0.2  [PLK1 -> SegB2.PLK2 (NodeNumber=3) [Cable Type=PowerlinkCable, Length=10, Version=1.0.0.3]; PLK2 -> SegB18.PLK1 (NodeNumber=3) [Cable Type=PowerlinkCable, Length=10, Version=1.0.0.3]; PLK3 -> X20HB2880.ETH2 (NodeNumber=3) [Cable Type=PowerlinkCable, Length=10, Version=1.0.0.3]]
  DriveConfiguration:
    McTypeID = LLMConfig
  DriveConfiguration/Segment:
    Shape = CIRCULAR_TO_STRAIGHT105
    SegmentReference = gSegB1
    SegmentSectorDirection = Positive
    ElongationCompensation = UseAssemblySetting
    StopReaction = UseAssemblySetting
    SpeedFilter = UseAssemblySetting
SegB10 : 8F1I01.BA2B.xxxx-1 v1.0.0.2  [PLK2 -> SegB9.PLK1 (NodeNumber=12) [Cable Type=PowerlinkCable, Length=10, Version=1.0.0.3]]
  DriveConfiguration:
    McTypeID = LLMConfig
  DriveConfiguration/Segment:
    Shape = CIRCULAR_TO_STRAIGHT105
    SegmentReference = gSegB10
    SegmentSectorDirection = Positive
    ElongationCompensation = UseAssemblySetting
    StopReaction = UseAssemblySetting
    SpeedFilter = UseAssemblySetting
SegB11 : 8F1I01.BB4B.xxxx-1 v1.0.0.2  [PLK1 -> SegB12.PLK2 (NodeNumber=11) [Cable Type=PowerlinkCable, Length=10, Version=1.0.0.3]]
  DriveConfiguration:
    McTypeID = LLMConfig
  DriveConfiguration/Segment:
    Shape = CIRCULAR
    SegmentReference = gSegB11
    SegmentSectorDirection = Positive
    ElongationCompensation = UseAssemblySetting
    StopReaction = UseAssemblySetting
    SpeedFilter = UseAssemblySetting
SegB12 : 8F1I01.BB4B.xxxx-1 v1.0.0.2  [PLK1 -> SegB13.PLK2 (NodeNumber=10) [Cable Type=PowerlinkCable, Length=10, Version=1.0.0.3]; PLK2 -> SegB11.PLK1 (NodeNumber=10) [Cable Type=PowerlinkCable, Length=10, Version=1.0.0.3]]
  DriveConfiguration:
    McTypeID = LLMConfig
  DriveConfiguration/Segment:
    Shape = CIRCULAR
    SegmentReference = gSegB12
    SegmentSectorDirection = Positive
    ElongationCompensation = UseAssemblySetting
    StopReaction = UseAssemblySetting
    SpeedFilter = UseAssemblySetting
SegB13 : 8F1I01.BB4B.xxxx-1 v1.0.0.2  [PLK1 -> SegB14.PLK2 (NodeNumber=9) [Cable Type=PowerlinkCable, Length=10, Version=1.0.0.3]; PLK2 -> SegB12.PLK1 (NodeNumber=9) [Cable Type=PowerlinkCable, Length=10, Version=1.0.0.3]]
  DriveConfiguration:
    McTypeID = LLMConfig
  DriveConfiguration/Segment:
    Shape = CIRCULAR
    SegmentReference = gSegB13
    SegmentSectorDirection = Positive
    ElongationCompensation = UseAssemblySetting
    StopReaction = UseAssemblySetting
    SpeedFilter = UseAssemblySetting
SegB14 : 8F1I01.AB2B.xxxx-1 v1.0.0.2  [PLK1 -> SegB15.PLK2 (NodeNumber=8) [Cable Type=PowerlinkCable, Length=10, Version=1.0.0.3]; PLK2 -> SegB13.PLK1 (NodeNumber=8) [Cable Type=PowerlinkCable, Length=10, Version=1.0.0.3]]
  DriveConfiguration:
    McTypeID = LLMConfig
  DriveConfiguration/Segment:
    Shape = STRAIGHT105_TO_CIRCULAR
    SegmentReference = gSegB14
    SegmentSectorDirection = Positive
    ElongationCompensation = UseAssemblySetting
    StopReaction = UseAssemblySetting
    SpeedFilter = UseAssemblySetting
SegB15 : 8F1I01.AB2B.xxxx-1 v1.0.0.2  [PLK1 -> SegB16.PLK2 (NodeNumber=7) [Cable Type=PowerlinkCable, Length=10, Version=1.0.0.3]; PLK2 -> SegB14.PLK1 (NodeNumber=7) [Cable Type=PowerlinkCable, Length=10, Version=1.0.0.3]]
  DriveConfiguration:
    McTypeID = LLMConfig
  DriveConfiguration/Segment:
    Shape = STRAIGHT105_TO_CIRCULAR
    SegmentReference = gSegB15
    SegmentSectorDirection = Positive
    ElongationCompensation = UseAssemblySetting
    StopReaction = UseAssemblySetting
    SpeedFilter = UseAssemblySetting
SegB16 : 8F1I01.BA2B.xxxx-1 v1.0.0.2  [PLK1 -> SegB17.PLK2 (NodeNumber=6) [Cable Type=PowerlinkCable, Length=10, Version=1.0.0.3]; PLK2 -> SegB15.PLK1 (NodeNumber=6) [Cable Type=PowerlinkCable, Length=10, Version=1.0.0.3]]
  DriveConfiguration:
    McTypeID = LLMConfig
  DriveConfiguration/Segment:
    Shape = CIRCULAR_TO_STRAIGHT105
    SegmentReference = gSegB16
    SegmentSectorDirection = Positive
    ElongationCompensation = UseAssemblySetting
    StopReaction = UseAssemblySetting
    SpeedFilter = UseAssemblySetting
SegB17 : 8F1I01.BA2B.xxxx-1 v1.0.0.2  [PLK1 -> SegB18.PLK2 (NodeNumber=5) [Cable Type=PowerlinkCable, Length=10, Version=1.0.0.3]; PLK2 -> SegB16.PLK1 (NodeNumber=5) [Cable Type=PowerlinkCable, Length=10, Version=1.0.0.3]]
  DriveConfiguration:
    McTypeID = LLMConfig
  DriveConfiguration/Segment:
    Shape = CIRCULAR_TO_STRAIGHT105
    SegmentReference = gSegB17
    SegmentSectorDirection = Positive
    ElongationCompensation = UseAssemblySetting
    StopReaction = UseAssemblySetting
    SpeedFilter = UseAssemblySetting
SegB18 : 8F1I01.AB2B.xxxx-1 v1.0.0.2  [PLK1 -> SegB1.PLK2 (NodeNumber=4) [Cable Type=PowerlinkCable, Length=10, Version=1.0.0.3]; PLK2 -> SegB17.PLK1 (NodeNumber=4) [Cable Type=PowerlinkCable, Length=10, Version=1.0.0.3]]
  DriveConfiguration:
    McTypeID = LLMConfig
  DriveConfiguration/Segment:
    Shape = STRAIGHT105_TO_CIRCULAR
    SegmentReference = gSegB18
    SegmentSectorDirection = Positive
    ElongationCompensation = UseAssemblySetting
    StopReaction = UseAssemblySetting
    SpeedFilter = UseAssemblySetting
SegB2 : 8F1I01.BB4B.xxxx-1 v1.0.0.2  [PLK1 -> SegB3.PLK2 (NodeNumber=13) [Cable Type=PowerlinkCable, Length=10, Version=1.0.0.3]; PLK2 -> SegB1.PLK1 (NodeNumber=13) [Cable Type=PowerlinkCable, Length=10, Version=1.0.0.3]]
  DriveConfiguration:
    McTypeID = LLMConfig
  DriveConfiguration/Segment:
    Shape = CIRCULAR
    SegmentReference = gSegB2
    SegmentSectorDirection = Positive
    ElongationCompensation = UseAssemblySetting
    StopReaction = UseAssemblySetting
    SpeedFilter = UseAssemblySetting
SegB3 : 8F1I01.BB4B.xxxx-1 v1.0.0.2  [PLK1 -> SegB4.PLK2 (NodeNumber=14) [Cable Type=PowerlinkCable, Length=10, Version=1.0.0.3]; PLK2 -> SegB2.PLK1 (NodeNumber=14) [Cable Type=PowerlinkCable, Length=10, Version=1.0.0.3]]
  DriveConfiguration:
    McTypeID = LLMConfig
  DriveConfiguration/Segment:
    Shape = CIRCULAR
    SegmentReference = gSegB3
    SegmentSectorDirection = Positive
    ElongationCompensation = UseAssemblySetting
    StopReaction = UseAssemblySetting
    SpeedFilter = UseAssemblySetting
SegB4 : 8F1I01.BB4B.xxxx-1 v1.0.0.2  [PLK1 -> SegB5.PLK2 (NodeNumber=15) [Cable Type=PowerlinkCable, Length=10, Version=1.0.0.3]; PLK2 -> SegB3.PLK1 (NodeNumber=15) [Cable Type=PowerlinkCable, Length=10, Version=1.0.0.3]]
  DriveConfiguration:
    McTypeID = LLMConfig
  DriveConfiguration/Segment:
    Shape = CIRCULAR
    SegmentReference = gSegB4
    SegmentSectorDirection = Positive
    ElongationCompensation = UseAssemblySetting
    StopReaction = UseAssemblySetting
    SpeedFilter = UseAssemblySetting
SegB5 : 8F1I01.AB2B.xxxx-1 v1.0.0.2  [PLK1 -> SegB6.PLK2 (NodeNumber=16) [Cable Type=PowerlinkCable, Length=10, Version=1.0.0.3]; PLK2 -> SegB4.PLK1 (NodeNumber=16) [Cable Type=PowerlinkCable, Length=10, Version=1.0.0.3]]
  DriveConfiguration:
    McTypeID = LLMConfig
  DriveConfiguration/Segment:
    Shape = STRAIGHT105_TO_CIRCULAR
    SegmentReference = gSegB5
    SegmentSectorDirection = Positive
    ElongationCompensation = UseAssemblySetting
    StopReaction = UseAssemblySetting
    SpeedFilter = UseAssemblySetting
SegB6 : 8F1I01.AB2B.xxxx-1 v1.0.0.2  [PLK1 -> SegB7.PLK2 (NodeNumber=17) [Cable Type=PowerlinkCable, Length=10, Version=1.0.0.3]; PLK2 -> SegB5.PLK1 (NodeNumber=17) [Cable Type=PowerlinkCable, Length=10, Version=1.0.0.3]]
  DriveConfiguration:
    McTypeID = LLMConfig
  DriveConfiguration/Segment:
    Shape = STRAIGHT105_TO_CIRCULAR
    SegmentReference = gSegB6
    SegmentSectorDirection = Positive
    ElongationCompensation = UseAssemblySetting
    StopReaction = UseAssemblySetting
    SpeedFilter = UseAssemblySetting
SegB7 : 8F1I01.BA2B.xxxx-1 v1.0.0.2  [PLK1 -> SegB8.PLK2 (NodeNumber=18) [Cable Type=PowerlinkCable, Length=10, Version=1.0.0.3]; PLK2 -> SegB6.PLK1 (NodeNumber=18) [Cable Type=PowerlinkCable, Length=10, Version=1.0.0.3]]
  DriveConfiguration:
    McTypeID = LLMConfig
  DriveConfiguration/Segment:
    Shape = CIRCULAR_TO_STRAIGHT105
    SegmentReference = gSegB7
    SegmentSectorDirection = Positive
    ElongationCompensation = UseAssemblySetting
    StopReaction = UseAssemblySetting
    SpeedFilter = UseAssemblySetting
SegB8 : 8F1I01.BA2B.xxxx-1 v1.0.0.2  [PLK1 -> SegB9.PLK2 (NodeNumber=20) [Cable Type=PowerlinkCable, Length=10, Version=1.0.0.3]; PLK2 -> SegB7.PLK1 (NodeNumber=20) [Cable Type=PowerlinkCable, Length=10, Version=1.0.0.3]]
  DriveConfiguration:
    McTypeID = LLMConfig
  DriveConfiguration/Segment:
    Shape = CIRCULAR_TO_STRAIGHT105
    SegmentReference = gSegB8
    SegmentSectorDirection = Positive
    ElongationCompensation = UseAssemblySetting
    StopReaction = UseAssemblySetting
    SpeedFilter = UseAssemblySetting
SegB9 : 8F1I01.AB2B.xxxx-1 v1.0.0.2  [PLK1 -> SegB10.PLK2 (NodeNumber=19) [Cable Type=PowerlinkCable, Length=10, Version=1.0.0.3]; PLK2 -> SegB8.PLK1 (NodeNumber=19) [Cable Type=PowerlinkCable, Length=10, Version=1.0.0.3]]
  DriveConfiguration:
    McTypeID = LLMConfig
  DriveConfiguration/Segment:
    Shape = STRAIGHT105_TO_CIRCULAR
    SegmentReference = gSegB9
    SegmentSectorDirection = Positive
    ElongationCompensation = UseAssemblySetting
    StopReaction = UseAssemblySetting
    SpeedFilter = UseAssemblySetting
X20BB80 : X20BB80 v1.1.0.0
X20BB81a : X20BB81 v1.1.0.0
  Connector IF1:
    ActivateX2X = 0
X20BC0083 : X20BC0083 v2.14.0.0  [PLK1 -> X20HB2880.ETH1 (NodeNumber=33) [Cable Type=PowerlinkCable, Length=10, Version=1.0.0.3]; SL -> X20BB80.SL1]
  Supervision = off
X20BM11 : X20BM11 v1.1.0.0  [X2X1 -> X20BB80.IF1]
X20BT9400 : X20BT9400 v1.3.0.0  [SS1 -> X20TB12b.SS; SL -> X20BM11.SL1]
  Supervision = off
X20CP3686X : X20CP3686X v1.6.2.0
  Connector IF2:
    ActivateDevice = 1
    Mode = Manual
    InternetAddress = 192.168.0.105
    SubnetMask = 255.255.255.0
    ActivateSnmp = 2
  Connector IF3:
    CycleTime = 2000
  ConfigurationID = mvDemoTrak_CP1685
  MotionLoggerSize = 2048000
  EnableUsbRemoteInstall = 1
  TimerDeviceType = EPLX2X
  TimerDevice = X20CP3686X.IF3
  TaskClassIdleTime = 2000
  Cyclic1Duration = 2000
  Cyclic1Tolerance = 0
  Cyclic2Duration = 10000
  Cyclic2Tolerance = 10000
  FileDevice1
  FileDeviceName1 = SvgData
  FileDevicePath1 = F:\web\SvgData
  FileDevice2
  FileDeviceName2 = Diagnosis
  FileDevicePath2 = F:\web\Diagnosis
  FileDevice3
  FileDeviceName3 = USER
  FileDevicePath3 = F:\
  FtpUser1
  FtpUsername1 = Admin
  FtpUserPassword1 = b2dkeklN0DR4HlzomfG8N5dlVtI3Hrgd5HBjTL6T4A4=  // pw: admin
  FtpUserSalt1 = LZ6GLOae
  FTPAccessRight1 = 0
  FTPdevice1 = ALL
  WebServerWebDir = F:\web  // default: web\
  ActivateOpcUa = 1
  OpcUaInformationModels_PV_Version = 1
X20HB2880 : X20HB2880 v1.2.0.0  [ETH1 -> X20BC0083.PLK1 [Cable Type=PowerlinkCable, Length=10, Version=1.0.0.3]; ETH2 -> SegB1.PLK3 [Cable Type=PowerlinkCable, Length=10, Version=1.0.0.3]; SS -> X20BB81a.SS1]
X20HB8880 : X20HB8880 v1.1.0.0  [ETH1 -> X20CP3686X.IF3 [Cable Type=PowerlinkCable, Length=10, Version=1.0.0.3]; ETH2 -> SegA1.PLK3 [Cable Type=PowerlinkCable, Length=10, Version=1.0.0.3]; SL -> X20BB81a.SL1]
X20PS9400 : X20PS9400 v1.8.0.0  [SS1 -> X20TB12.SS; PS -> X20BB81a.PS1]
  Supervision = off
X20PS9400a : X20PS9400 v1.8.0.0  [SS1 -> X20TB12a.SS; PS -> X20BB80.PS1]
  Supervision = off
X20TB12 : X20TB12 v1.0.0.0
X20TB12a : X20TB12 v1.0.0.0
X20TB12b : X20TB12 v1.0.0.0
```

## Configuration Config1

CPU 5PC900.TS17-00, AutomationRuntime D4.93, Build 6.3.0, Safety 0.0, Vc 

### Task classes (Cpu.sw)
```
Cyclic#1 (cycle 2000 us, tolerance 0 us):
  TrakInit <- Trak.TrakInit.prg
Cyclic#2 (cycle 10000 us, tolerance 10000 us):
  AssCtrl <- Trak.AssCtrl.prg
  AlarmXTask <- VisuPackage.AlarmXTask.prg
  VisuTask <- VisuPackage.VisuTask.prg
Cyclic#4:
  SegCtrl <- Trak.SegCtrl.prg
DataObjects: McAcpSys
NcDataObjects: mcdrivelog
Binaries: McAcpSim, FWRules, arcoal, arsvcreg, TCData, McAcpDrv, mCoWebSc, mvLoader, arflatprv, udbdef, TCLang, iomap, Config_1, arconfig, asfw, ashwac, sysconf, User, Settings, Role, ashwd, Config_4, Config_3, Config_2, Config, CfgAlHist, TC, CfgAlList
Libraries: McBase, CoTrace, AsZip, FileIO, runtime, McAxis, McAcpTrak, MpBase, TrakLib, standard, AsBrStr, sys_lib, brsystem, astime, ArEventLog, DataObj, AsHttp, MpServer, TrakDiag, AsArSdm, powerlnk, arssl, asieccon, mpalarmx, aruser
```

### Hardware
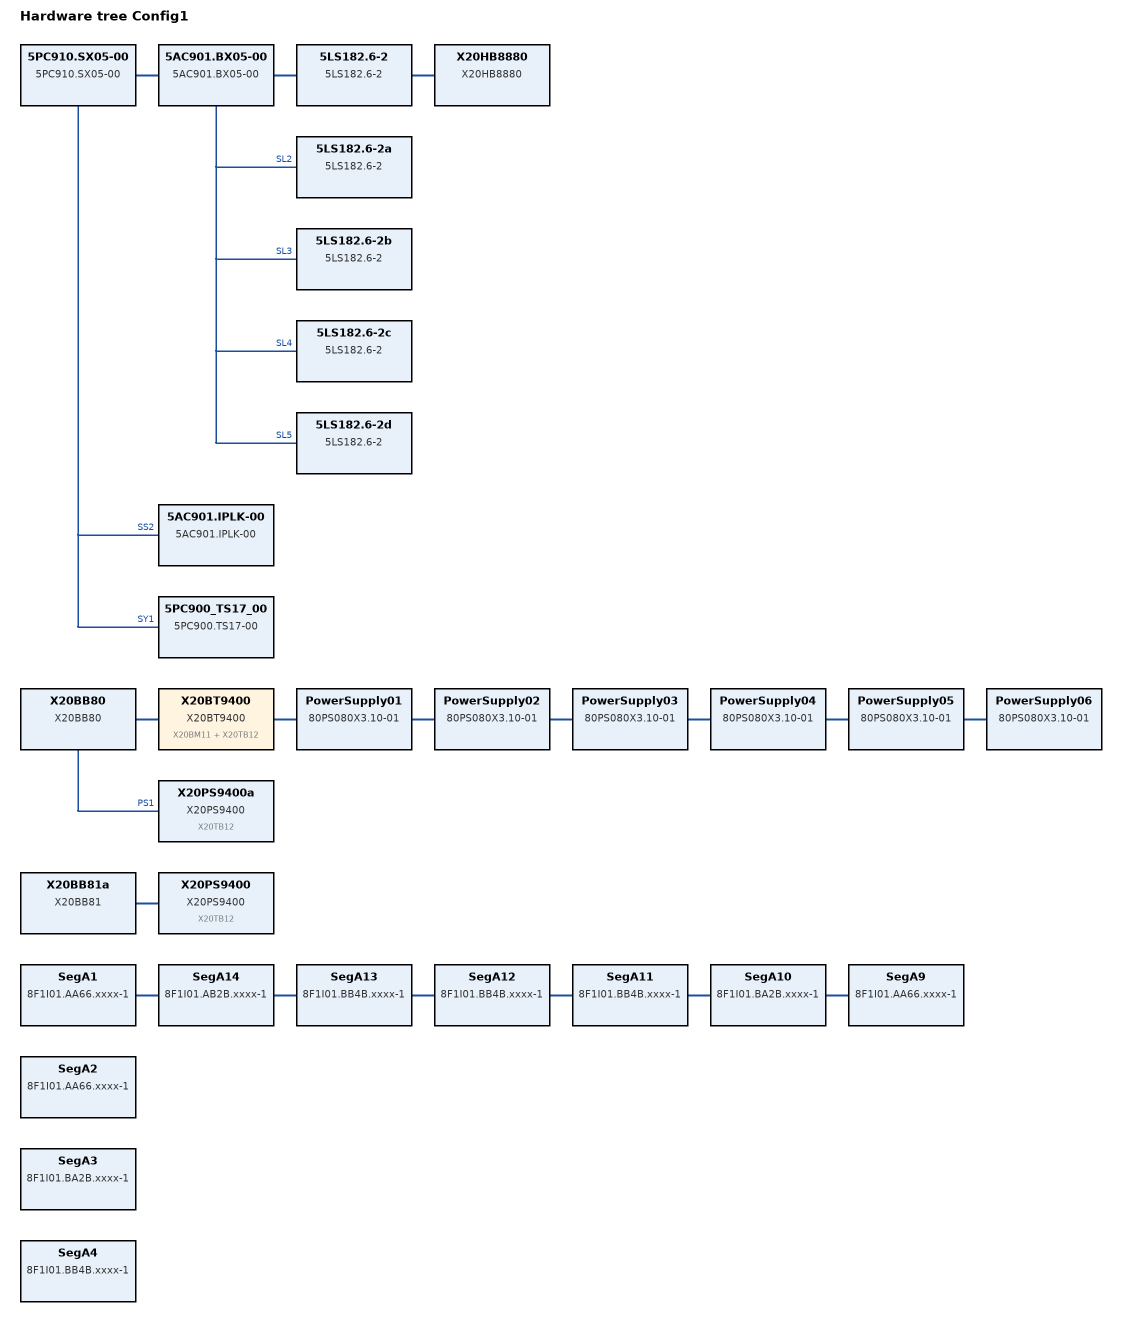
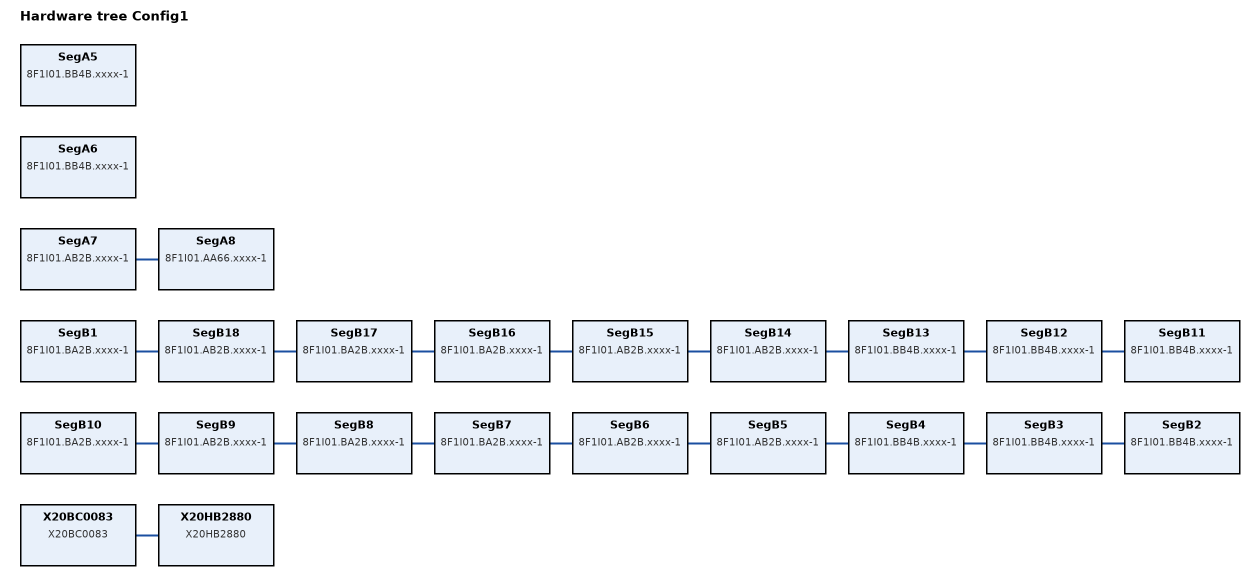
```
5AC901.BX05-00 : 5AC901.BX05-00 v1.0.1.0  [SY -> 5PC910.SX05-00.SY3]
5AC901.IPLK-00 : 5AC901.IPLK-00 v1.8.0.1 (Disabled=true)  [SS -> 5PC910.SX05-00.SS2]
  Connector IF1 (Disabled=true)
5LS182.6-2 : 5LS182.6-2 v1.9.0.0  [SL -> 5AC901.BX05-00.SL1]
  Connector IF1:
    EplHostName = mvdemotrak
    NodeDefinition = Software
    HostName = mvdemotrak
5LS182.6-2a : 5LS182.6-2 v1.9.0.0 (Disabled=true)  [SL -> 5AC901.BX05-00.SL2]
  Connector IF1 (Disabled=true)
    EplHostName = mvdemotrak
    HostName = mvdemotrak
5LS182.6-2b : 5LS182.6-2 v1.9.0.0 (Disabled=true)  [SL -> 5AC901.BX05-00.SL3]
  Connector IF1 (Disabled=true)
    EplHostName = mvdemotrak
    HostName = mvdemotrak
5LS182.6-2c : 5LS182.6-2 v1.9.0.0 (Disabled=true)  [SL -> 5AC901.BX05-00.SL4]
  Connector IF1 (Disabled=true)
    EplHostName = mvdemotrak
    HostName = mvdemotrak
5LS182.6-2d : 5LS182.6-2 v1.9.0.0 (Disabled=true)  [SL -> 5AC901.BX05-00.SL5]
  Connector IF1 (Disabled=true)
    EplHostName = mvdemotrak
    HostName = mvdemotrak
5PC900_TS17_00 : 5PC900.TS17-00 v2.1.0.0  [SY -> 5PC910.SX05-00.SY1]
  ConfigurationID = TrakDemo_Config1
  MotionLoggerSize = 2048000
  TaskClassIdleTime = 3000
  Cyclic1Duration = 2000
  Cyclic1Tolerance = 0
  Cyclic2Duration = 10000
  Cyclic2Tolerance = 10000
  FileDevice1
  FileDeviceName1 = SvgData
  FileDevicePath1 = F:\web\SvgData
  FileDevice2
  FileDeviceName2 = Diagnosis
  FileDevicePath2 = F:\web\Diagnosis
  FileDevice3
  FileDeviceName3 = USER
  FileDevicePath3 = F:\
  EthernetHostName = mvdemotrak
  EthernetDefaultGateway = 10.49.40.1
  FtpUser1
  FtpUsername1 = admin
  FtpUserPassword1 = 1eFk4bv95gGd/YhutE0/XT32p+eqiGHSQm0YwzXwS3M=
  FtpUserSalt1 = in5n/jXa
  FTPAccessRight1 = 0
  FTPdevice1 = ALL
  WebServerWebDir = F:\web\
  ActivateOpcUa = 1
  OpcUaInformationModels_PV_Version = 1
5PC910.SX05-00 : 5PC910.SX05-00 v2.1.0.0
  Connector IF1:
    AssignedOperatingSystem = ARemb
  Connector IF3:
    AssignedOperatingSystem = ARemb
    ActivateDevice = 1
    HostName = mvdemotrak
    Mode = Manual
    InternetAddress = 10.49.40.236
    SubnetMask = 255.255.255.0
    ActivateSnmp = 2
  Connector IF4:
    AssignedOperatingSystem = ARemb
    ActivateDevice = 1
    HostName = mvdemotrak
    Mode = Manual
    InternetAddress = 172.16.0.100
    SubnetMask = 255.255.255.0
    ActivateIna = 0
  Connector IF5:
    AssignedOperatingSystem = ARemb
  Connector IF6:
    AssignedOperatingSystem = ARemb
  Connector IF7:
    AssignedOperatingSystem = ARemb
  Connector IF8:
    AssignedOperatingSystem = ARemb
  Connector IF9:
    AssignedOperatingSystem = ARemb
PowerSupply01 : 80PS080X3.10-01 v1.5.0.0  [X2X1 -> X20BT9400.X2X1 [Cable Type=X2XCable, Length=10, Version=1.0.0.3]]
  Supervision = off
PowerSupply02 : 80PS080X3.10-01 v1.5.0.0  [X2X1 -> PowerSupply01.X2X2 [Cable Type=X2XCable, Length=10, Version=1.0.0.3]]
  Supervision = off
PowerSupply03 : 80PS080X3.10-01 v1.5.0.0  [X2X1 -> PowerSupply02.X2X2 [Cable Type=X2XCable, Length=10, Version=1.0.0.3]]
  Supervision = off
PowerSupply04 : 80PS080X3.10-01 v1.5.0.0  [X2X1 -> PowerSupply03.X2X2 [Cable Type=X2XCable, Length=10, Version=1.0.0.3]]
  Supervision = off
PowerSupply05 : 80PS080X3.10-01 v1.5.0.0  [X2X1 -> PowerSupply04.X2X2 [Cable Type=X2XCable, Length=10, Version=1.0.0.3]]
  Supervision = off
PowerSupply06 : 80PS080X3.10-01 v1.5.0.0  [X2X1 -> PowerSupply05.X2X2 [Cable Type=X2XCable, Length=10, Version=1.0.0.3]]
  Supervision = off
SegA1 : 8F1I01.AA66.xxxx-1 v1.0.0.2  [PLK1 -> SegA2.PLK2 (NodeNumber=1) [Cable Type=PowerlinkCable, Length=10, Version=1.0.0.3]; PLK2 -> SegA14.PLK1 (NodeNumber=1) [Cable Type=PowerlinkCable, Length=10, Version=1.0.0.3]; PLK3 -> X20HB8880.ETH2 (NodeNumber=1) [Cable Type=PowerlinkCable, Length=10, Version=1.0.0.3]]
  DriveConfiguration:
    McTypeID = LLMConfig
  DriveConfiguration/Segment:
    Shape = STRAIGHT660
    SegmentReference = gSegA1
    SegmentSectorDirection = Positive
    ElongationCompensation = UseAssemblySetting
    StopReaction = UseAssemblySetting
    SpeedFilter = UseAssemblySetting
SegA10 : 8F1I01.BA2B.xxxx-1 v1.0.0.2  [PLK1 -> SegA11.PLK2 (NodeNumber=25) [Cable Type=PowerlinkCable, Length=10, Version=1.0.0.3]; PLK2 -> SegA9.PLK1 (NodeNumber=25) [Cable Type=PowerlinkCable, Length=10, Version=1.0.0.3]]
  DriveConfiguration:
    McTypeID = LLMConfig
  DriveConfiguration/Segment:
    Shape = CIRCULAR_TO_STRAIGHT105
    SegmentReference = gSegA10
    SegmentSectorDirection = Positive
    ElongationCompensation = UseAssemblySetting
    StopReaction = UseAssemblySetting
    SpeedFilter = UseAssemblySetting
SegA11 : 8F1I01.BB4B.xxxx-1 v1.0.0.2  [PLK1 -> SegA12.PLK2 (NodeNumber=24) [Cable Type=PowerlinkCable, Length=10, Version=1.0.0.3]; PLK2 -> SegA10.PLK1 (NodeNumber=24) [Cable Type=PowerlinkCable, Length=10, Version=1.0.0.3]]
  DriveConfiguration:
    McTypeID = LLMConfig
  DriveConfiguration/Segment:
    Shape = CIRCULAR
    SegmentReference = gSegA11
    SegmentSectorDirection = Positive
    ElongationCompensation = UseAssemblySetting
    StopReaction = UseAssemblySetting
    SpeedFilter = UseAssemblySetting
SegA12 : 8F1I01.BB4B.xxxx-1 v1.0.0.2  [PLK1 -> SegA13.PLK2 (NodeNumber=23) [Cable Type=PowerlinkCable, Length=10, Version=1.0.0.3]; PLK2 -> SegA11.PLK1 (NodeNumber=23) [Cable Type=PowerlinkCable, Length=10, Version=1.0.0.3]]
  DriveConfiguration:
    McTypeID = LLMConfig
  DriveConfiguration/Segment:
    Shape = CIRCULAR
    SegmentReference = gSegA12
    SegmentSectorDirection = Positive
    ElongationCompensation = UseAssemblySetting
    StopReaction = UseAssemblySetting
    SpeedFilter = UseAssemblySetting
SegA13 : 8F1I01.BB4B.xxxx-1 v1.0.0.2  [PLK1 -> SegA14.PLK2 (NodeNumber=22) [Cable Type=PowerlinkCable, Length=10, Version=1.0.0.3]; PLK2 -> SegA12.PLK1 (NodeNumber=22) [Cable Type=PowerlinkCable, Length=10, Version=1.0.0.3]]
  DriveConfiguration:
    McTypeID = LLMConfig
  DriveConfiguration/Segment:
    Shape = CIRCULAR
    SegmentReference = gSegA13
    SegmentSectorDirection = Positive
    ElongationCompensation = UseAssemblySetting
    StopReaction = UseAssemblySetting
    SpeedFilter = UseAssemblySetting
SegA14 : 8F1I01.AB2B.xxxx-1 v1.0.0.2  [PLK1 -> SegA1.PLK2 (NodeNumber=21) [Cable Type=PowerlinkCable, Length=10, Version=1.0.0.3]; PLK2 -> SegA13.PLK1 (NodeNumber=21) [Cable Type=PowerlinkCable, Length=10, Version=1.0.0.3]]
  DriveConfiguration:
    McTypeID = LLMConfig
  DriveConfiguration/Segment:
    Shape = STRAIGHT105_TO_CIRCULAR
    SegmentReference = gSegA14
    SegmentSectorDirection = Positive
    ElongationCompensation = UseAssemblySetting
    StopReaction = UseAssemblySetting
    SpeedFilter = UseAssemblySetting
SegA2 : 8F1I01.AA66.xxxx-1 v1.0.0.2  [PLK1 -> SegA3.PLK2 (NodeNumber=2) [Cable Type=PowerlinkCable, Length=10, Version=1.0.0.3]; PLK2 -> SegA1.PLK1 (NodeNumber=2) [Cable Type=PowerlinkCable, Length=10, Version=1.0.0.3]]
  DriveConfiguration:
    McTypeID = LLMConfig
  DriveConfiguration/Segment:
    Shape = STRAIGHT660
    SegmentReference = gSegA2
    SegmentSectorDirection = Positive
    ElongationCompensation = UseAssemblySetting
    StopReaction = UseAssemblySetting
    SpeedFilter = UseAssemblySetting
SegA3 : 8F1I01.BA2B.xxxx-1 v1.0.0.2  [PLK1 -> SegA4.PLK2 (NodeNumber=27) [Cable Type=PowerlinkCable, Length=10, Version=1.0.0.3]; PLK2 -> SegA2.PLK1 (NodeNumber=27) [Cable Type=PowerlinkCable, Length=10, Version=1.0.0.3]]
  DriveConfiguration:
    McTypeID = LLMConfig
  DriveConfiguration/Segment:
    Shape = CIRCULAR_TO_STRAIGHT105
    SegmentReference = gSegA3
    SegmentSectorDirection = Positive
    ElongationCompensation = UseAssemblySetting
    StopReaction = UseAssemblySetting
    SpeedFilter = UseAssemblySetting
SegA4 : 8F1I01.BB4B.xxxx-1 v1.0.0.2  [PLK1 -> SegA5.PLK2 (NodeNumber=28) [Cable Type=PowerlinkCable, Length=10, Version=1.0.0.3]; PLK2 -> SegA3.PLK1 (NodeNumber=28) [Cable Type=PowerlinkCable, Length=10, Version=1.0.0.3]]
  DriveConfiguration:
    McTypeID = LLMConfig
  DriveConfiguration/Segment:
    Shape = CIRCULAR
    SegmentReference = gSegA4
    SegmentSectorDirection = Positive
    ElongationCompensation = UseAssemblySetting
    StopReaction = UseAssemblySetting
    SpeedFilter = UseAssemblySetting
SegA5 : 8F1I01.BB4B.xxxx-1 v1.0.0.2  [PLK1 -> SegA6.PLK2 (NodeNumber=29) [Cable Type=PowerlinkCable, Length=10, Version=1.0.0.3]; PLK2 -> SegA4.PLK1 (NodeNumber=29) [Cable Type=PowerlinkCable, Length=10, Version=1.0.0.3]]
  DriveConfiguration:
    McTypeID = LLMConfig
  DriveConfiguration/Segment:
    Shape = CIRCULAR
    SegmentReference = gSegA5
    SegmentSectorDirection = Positive
    ElongationCompensation = UseAssemblySetting
    StopReaction = UseAssemblySetting
    SpeedFilter = UseAssemblySetting
SegA6 : 8F1I01.BB4B.xxxx-1 v1.0.0.2  [PLK1 -> SegA7.PLK2 (NodeNumber=30) [Cable Type=PowerlinkCable, Length=10, Version=1.0.0.3]; PLK2 -> SegA5.PLK1 (NodeNumber=30) [Cable Type=PowerlinkCable, Length=10, Version=1.0.0.3]]
  DriveConfiguration:
    McTypeID = LLMConfig
  DriveConfiguration/Segment:
    Shape = CIRCULAR
    SegmentReference = gSegA6
    SegmentSectorDirection = Positive
    ElongationCompensation = UseAssemblySetting
    StopReaction = UseAssemblySetting
    SpeedFilter = UseAssemblySetting
SegA7 : 8F1I01.AB2B.xxxx-1 v1.0.0.2  [PLK1 -> SegA8.PLK2 (NodeNumber=31) [Cable Type=PowerlinkCable, Length=10, Version=1.0.0.3]; PLK2 -> SegA6.PLK1 (NodeNumber=31) [Cable Type=PowerlinkCable, Length=10, Version=1.0.0.3]]
  DriveConfiguration:
    McTypeID = LLMConfig
  DriveConfiguration/Segment:
    Shape = STRAIGHT105_TO_CIRCULAR
    SegmentReference = gSegA7
    SegmentSectorDirection = Positive
    ElongationCompensation = UseAssemblySetting
    StopReaction = UseAssemblySetting
    SpeedFilter = UseAssemblySetting
SegA8 : 8F1I01.AA66.xxxx-1 v1.0.0.2  [PLK2 -> SegA7.PLK1 (NodeNumber=32) [Cable Type=PowerlinkCable, Length=10, Version=1.0.0.3]]
  DriveConfiguration:
    McTypeID = LLMConfig
  DriveConfiguration/Segment:
    Shape = STRAIGHT660
    SegmentReference = gSegA8
    SegmentSectorDirection = Positive
    ElongationCompensation = UseAssemblySetting
    StopReaction = UseAssemblySetting
    SpeedFilter = UseAssemblySetting
SegA9 : 8F1I01.AA66.xxxx-1 v1.0.0.2  [PLK1 -> SegA10.PLK2 (NodeNumber=26) [Cable Type=PowerlinkCable, Length=10, Version=1.0.0.3]]
  DriveConfiguration:
    McTypeID = LLMConfig
  DriveConfiguration/Segment:
    Shape = STRAIGHT660
    SegmentReference = gSegA9
    SegmentSectorDirection = Positive
    ElongationCompensation = UseAssemblySetting
    StopReaction = UseAssemblySetting
    SpeedFilter = UseAssemblySetting
SegB1 : 8F1I01.BA2B.xxxx-1 v1.0.0.2  [PLK1 -> SegB2.PLK2 (NodeNumber=3) [Cable Type=PowerlinkCable, Length=10, Version=1.0.0.3]; PLK2 -> SegB18.PLK1 (NodeNumber=3) [Cable Type=PowerlinkCable, Length=10, Version=1.0.0.3]; PLK3 -> X20HB2880.ETH2 (NodeNumber=3) [Cable Type=PowerlinkCable, Length=10, Version=1.0.0.3]]
  DriveConfiguration:
    McTypeID = LLMConfig
  DriveConfiguration/Segment:
    Shape = CIRCULAR_TO_STRAIGHT105
    SegmentReference = gSegB1
    SegmentSectorDirection = Positive
    ElongationCompensation = UseAssemblySetting
    StopReaction = UseAssemblySetting
    SpeedFilter = UseAssemblySetting
SegB10 : 8F1I01.BA2B.xxxx-1 v1.0.0.2  [PLK2 -> SegB9.PLK1 (NodeNumber=12) [Cable Type=PowerlinkCable, Length=10, Version=1.0.0.3]]
  DriveConfiguration:
    McTypeID = LLMConfig
  DriveConfiguration/Segment:
    Shape = CIRCULAR_TO_STRAIGHT105
    SegmentReference = gSegB10
    SegmentSectorDirection = Positive
    ElongationCompensation = UseAssemblySetting
    StopReaction = UseAssemblySetting
    SpeedFilter = UseAssemblySetting
SegB11 : 8F1I01.BB4B.xxxx-1 v1.0.0.2  [PLK1 -> SegB12.PLK2 (NodeNumber=11) [Cable Type=PowerlinkCable, Length=10, Version=1.0.0.3]]
  DriveConfiguration:
    McTypeID = LLMConfig
  DriveConfiguration/Segment:
    Shape = CIRCULAR
    SegmentReference = gSegB11
    SegmentSectorDirection = Positive
    ElongationCompensation = UseAssemblySetting
    StopReaction = UseAssemblySetting
    SpeedFilter = UseAssemblySetting
SegB12 : 8F1I01.BB4B.xxxx-1 v1.0.0.2  [PLK1 -> SegB13.PLK2 (NodeNumber=10) [Cable Type=PowerlinkCable, Length=10, Version=1.0.0.3]; PLK2 -> SegB11.PLK1 (NodeNumber=10) [Cable Type=PowerlinkCable, Length=10, Version=1.0.0.3]]
  DriveConfiguration:
    McTypeID = LLMConfig
  DriveConfiguration/Segment:
    Shape = CIRCULAR
    SegmentReference = gSegB12
    SegmentSectorDirection = Positive
    ElongationCompensation = UseAssemblySetting
    StopReaction = UseAssemblySetting
    SpeedFilter = UseAssemblySetting
SegB13 : 8F1I01.BB4B.xxxx-1 v1.0.0.2  [PLK1 -> SegB14.PLK2 (NodeNumber=9) [Cable Type=PowerlinkCable, Length=10, Version=1.0.0.3]; PLK2 -> SegB12.PLK1 (NodeNumber=9) [Cable Type=PowerlinkCable, Length=10, Version=1.0.0.3]]
  DriveConfiguration:
    McTypeID = LLMConfig
  DriveConfiguration/Segment:
    Shape = CIRCULAR
    SegmentReference = gSegB13
    SegmentSectorDirection = Positive
    ElongationCompensation = UseAssemblySetting
    StopReaction = UseAssemblySetting
    SpeedFilter = UseAssemblySetting
SegB14 : 8F1I01.AB2B.xxxx-1 v1.0.0.2  [PLK1 -> SegB15.PLK2 (NodeNumber=8) [Cable Type=PowerlinkCable, Length=10, Version=1.0.0.3]; PLK2 -> SegB13.PLK1 (NodeNumber=8) [Cable Type=PowerlinkCable, Length=10, Version=1.0.0.3]]
  DriveConfiguration:
    McTypeID = LLMConfig
  DriveConfiguration/Segment:
    Shape = STRAIGHT105_TO_CIRCULAR
    SegmentReference = gSegB14
    SegmentSectorDirection = Positive
    ElongationCompensation = UseAssemblySetting
    StopReaction = UseAssemblySetting
    SpeedFilter = UseAssemblySetting
SegB15 : 8F1I01.AB2B.xxxx-1 v1.0.0.2  [PLK1 -> SegB16.PLK2 (NodeNumber=7) [Cable Type=PowerlinkCable, Length=10, Version=1.0.0.3]; PLK2 -> SegB14.PLK1 (NodeNumber=7) [Cable Type=PowerlinkCable, Length=10, Version=1.0.0.3]]
  DriveConfiguration:
    McTypeID = LLMConfig
  DriveConfiguration/Segment:
    Shape = STRAIGHT105_TO_CIRCULAR
    SegmentReference = gSegB15
    SegmentSectorDirection = Positive
    ElongationCompensation = UseAssemblySetting
    StopReaction = UseAssemblySetting
    SpeedFilter = UseAssemblySetting
SegB16 : 8F1I01.BA2B.xxxx-1 v1.0.0.2  [PLK1 -> SegB17.PLK2 (NodeNumber=6) [Cable Type=PowerlinkCable, Length=10, Version=1.0.0.3]; PLK2 -> SegB15.PLK1 (NodeNumber=6) [Cable Type=PowerlinkCable, Length=10, Version=1.0.0.3]]
  DriveConfiguration:
    McTypeID = LLMConfig
  DriveConfiguration/Segment:
    Shape = CIRCULAR_TO_STRAIGHT105
    SegmentReference = gSegB16
    SegmentSectorDirection = Positive
    ElongationCompensation = UseAssemblySetting
    StopReaction = UseAssemblySetting
    SpeedFilter = UseAssemblySetting
SegB17 : 8F1I01.BA2B.xxxx-1 v1.0.0.2  [PLK1 -> SegB18.PLK2 (NodeNumber=5) [Cable Type=PowerlinkCable, Length=10, Version=1.0.0.3]; PLK2 -> SegB16.PLK1 (NodeNumber=5) [Cable Type=PowerlinkCable, Length=10, Version=1.0.0.3]]
  DriveConfiguration:
    McTypeID = LLMConfig
  DriveConfiguration/Segment:
    Shape = CIRCULAR_TO_STRAIGHT105
    SegmentReference = gSegB17
    SegmentSectorDirection = Positive
    ElongationCompensation = UseAssemblySetting
    StopReaction = UseAssemblySetting
    SpeedFilter = UseAssemblySetting
SegB18 : 8F1I01.AB2B.xxxx-1 v1.0.0.2  [PLK1 -> SegB1.PLK2 (NodeNumber=4) [Cable Type=PowerlinkCable, Length=10, Version=1.0.0.3]; PLK2 -> SegB17.PLK1 (NodeNumber=4) [Cable Type=PowerlinkCable, Length=10, Version=1.0.0.3]]
  DriveConfiguration:
    McTypeID = LLMConfig
  DriveConfiguration/Segment:
    Shape = STRAIGHT105_TO_CIRCULAR
    SegmentReference = gSegB18
    SegmentSectorDirection = Positive
    ElongationCompensation = UseAssemblySetting
    StopReaction = UseAssemblySetting
    SpeedFilter = UseAssemblySetting
SegB2 : 8F1I01.BB4B.xxxx-1 v1.0.0.2  [PLK1 -> SegB3.PLK2 (NodeNumber=13) [Cable Type=PowerlinkCable, Length=10, Version=1.0.0.3]; PLK2 -> SegB1.PLK1 (NodeNumber=13) [Cable Type=PowerlinkCable, Length=10, Version=1.0.0.3]]
  DriveConfiguration:
    McTypeID = LLMConfig
  DriveConfiguration/Segment:
    Shape = CIRCULAR
    SegmentReference = gSegB2
    SegmentSectorDirection = Positive
    ElongationCompensation = UseAssemblySetting
    StopReaction = UseAssemblySetting
    SpeedFilter = UseAssemblySetting
SegB3 : 8F1I01.BB4B.xxxx-1 v1.0.0.2  [PLK1 -> SegB4.PLK2 (NodeNumber=14) [Cable Type=PowerlinkCable, Length=10, Version=1.0.0.3]; PLK2 -> SegB2.PLK1 (NodeNumber=14) [Cable Type=PowerlinkCable, Length=10, Version=1.0.0.3]]
  DriveConfiguration:
    McTypeID = LLMConfig
  DriveConfiguration/Segment:
    Shape = CIRCULAR
    SegmentReference = gSegB3
    SegmentSectorDirection = Positive
    ElongationCompensation = UseAssemblySetting
    StopReaction = UseAssemblySetting
    SpeedFilter = UseAssemblySetting
SegB4 : 8F1I01.BB4B.xxxx-1 v1.0.0.2  [PLK1 -> SegB5.PLK2 (NodeNumber=15) [Cable Type=PowerlinkCable, Length=10, Version=1.0.0.3]; PLK2 -> SegB3.PLK1 (NodeNumber=15) [Cable Type=PowerlinkCable, Length=10, Version=1.0.0.3]]
  DriveConfiguration:
    McTypeID = LLMConfig
  DriveConfiguration/Segment:
    Shape = CIRCULAR
    SegmentReference = gSegB4
    SegmentSectorDirection = Positive
    ElongationCompensation = UseAssemblySetting
    StopReaction = UseAssemblySetting
    SpeedFilter = UseAssemblySetting
SegB5 : 8F1I01.AB2B.xxxx-1 v1.0.0.2  [PLK1 -> SegB6.PLK2 (NodeNumber=16) [Cable Type=PowerlinkCable, Length=10, Version=1.0.0.3]; PLK2 -> SegB4.PLK1 (NodeNumber=16) [Cable Type=PowerlinkCable, Length=10, Version=1.0.0.3]]
  DriveConfiguration:
    McTypeID = LLMConfig
  DriveConfiguration/Segment:
    Shape = STRAIGHT105_TO_CIRCULAR
    SegmentReference = gSegB5
    SegmentSectorDirection = Positive
    ElongationCompensation = UseAssemblySetting
    StopReaction = UseAssemblySetting
    SpeedFilter = UseAssemblySetting
SegB6 : 8F1I01.AB2B.xxxx-1 v1.0.0.2  [PLK1 -> SegB7.PLK2 (NodeNumber=17) [Cable Type=PowerlinkCable, Length=10, Version=1.0.0.3]; PLK2 -> SegB5.PLK1 (NodeNumber=17) [Cable Type=PowerlinkCable, Length=10, Version=1.0.0.3]]
  DriveConfiguration:
    McTypeID = LLMConfig
  DriveConfiguration/Segment:
    Shape = STRAIGHT105_TO_CIRCULAR
    SegmentReference = gSegB6
    SegmentSectorDirection = Positive
    ElongationCompensation = UseAssemblySetting
    StopReaction = UseAssemblySetting
    SpeedFilter = UseAssemblySetting
SegB7 : 8F1I01.BA2B.xxxx-1 v1.0.0.2  [PLK1 -> SegB8.PLK2 (NodeNumber=18) [Cable Type=PowerlinkCable, Length=10, Version=1.0.0.3]; PLK2 -> SegB6.PLK1 (NodeNumber=18) [Cable Type=PowerlinkCable, Length=10, Version=1.0.0.3]]
  DriveConfiguration:
    McTypeID = LLMConfig
  DriveConfiguration/Segment:
    Shape = CIRCULAR_TO_STRAIGHT105
    SegmentReference = gSegB7
    SegmentSectorDirection = Positive
    ElongationCompensation = UseAssemblySetting
    StopReaction = UseAssemblySetting
    SpeedFilter = UseAssemblySetting
SegB8 : 8F1I01.BA2B.xxxx-1 v1.0.0.2  [PLK1 -> SegB9.PLK2 (NodeNumber=20) [Cable Type=PowerlinkCable, Length=10, Version=1.0.0.3]; PLK2 -> SegB7.PLK1 (NodeNumber=20) [Cable Type=PowerlinkCable, Length=10, Version=1.0.0.3]]
  DriveConfiguration:
    McTypeID = LLMConfig
  DriveConfiguration/Segment:
    Shape = CIRCULAR_TO_STRAIGHT105
    SegmentReference = gSegB8
    SegmentSectorDirection = Positive
    ElongationCompensation = UseAssemblySetting
    StopReaction = UseAssemblySetting
    SpeedFilter = UseAssemblySetting
SegB9 : 8F1I01.AB2B.xxxx-1 v1.0.0.2  [PLK1 -> SegB10.PLK2 (NodeNumber=19) [Cable Type=PowerlinkCable, Length=10, Version=1.0.0.3]; PLK2 -> SegB8.PLK1 (NodeNumber=19) [Cable Type=PowerlinkCable, Length=10, Version=1.0.0.3]]
  DriveConfiguration:
    McTypeID = LLMConfig
  DriveConfiguration/Segment:
    Shape = STRAIGHT105_TO_CIRCULAR
    SegmentReference = gSegB9
    SegmentSectorDirection = Positive
    ElongationCompensation = UseAssemblySetting
    StopReaction = UseAssemblySetting
    SpeedFilter = UseAssemblySetting
X20BB80 : X20BB80 v1.1.0.0
X20BB81a : X20BB81 v1.1.0.0
  Connector IF1:
    ActivateX2X = 0
X20BC0083 : X20BC0083 v2.14.0.0  [PLK1 -> X20HB2880.ETH1 (NodeNumber=33) [Cable Type=PowerlinkCable, Length=10, Version=1.0.0.3]; SL -> X20BB80.SL1]
  Supervision = off
X20BM11 : X20BM11 v1.1.0.0  [X2X1 -> X20BB80.IF1]
X20BT9400 : X20BT9400 v1.3.0.0  [SS1 -> X20TB12b.SS; SL -> X20BM11.SL1]
  Supervision = off
X20HB2880 : X20HB2880 v1.2.0.0  [ETH1 -> X20BC0083.PLK1 [Cable Type=PowerlinkCable, Length=10, Version=1.0.0.3]; ETH2 -> SegB1.PLK3 [Cable Type=PowerlinkCable, Length=10, Version=1.0.0.3]; SS -> X20BB81a.SS1]
X20HB8880 : X20HB8880 v1.1.0.0  [ETH1 -> 5LS182.6-2.IF1 [Cable Type=PowerlinkCable, Length=10, Version=1.0.0.3]; ETH2 -> SegA1.PLK3 [Cable Type=PowerlinkCable, Length=10, Version=1.0.0.3]; SL -> X20BB81a.SL1]
X20PS9400 : X20PS9400 v1.8.0.0  [SS1 -> X20TB12.SS; PS -> X20BB81a.PS1]
  Supervision = off
X20PS9400a : X20PS9400 v1.8.0.0  [SS1 -> X20TB12a.SS; PS -> X20BB80.PS1]
  Supervision = off
X20TB12 : X20TB12 v1.0.0.0
X20TB12a : X20TB12 v1.0.0.0
X20TB12b : X20TB12 v1.0.0.0
```

### Config.mappmotioncfg - 5PC900_TS17_00/mappMotion/Config.mappmotioncfg
```
Element MappMotionConfiguration (Type=mappmotioncfg)
  Processing:
    ProcessingTaskClass = 1
  SharedAlarms:
    Assembly = MpAlarmX
    Segment = MpAlarmX
      mapp.AlarmX.Core.Configuration:
        [3]:
          Code = 1100
          Severity = 100
    Sector = MpAlarmX
    Shuttle = MpAlarmX
      mapp.AlarmX.Core.Configuration:
        [3]:
          Code = 2100
          Severity = 100
```

### Config_1.assembly - 5PC900_TS17_00/mappMotion/Config_1.assembly
```
Element gAssembly_1 (Type=assembly)
  Tracks:
    TrackSeparation = 0.030
    Track[1]:
      Segments:
        SegmentRef[1] = gSegA1
        SegmentRef[2] = gSegA14
        SegmentRef[3] = gSegA13
        SegmentRef[4] = gSegA12
        SegmentRef[5] = gSegA11
        SegmentRef[6] = gSegA10
        SegmentRef[7] = gSegA9
        SegmentRef[8] = gSegA8
        SegmentRef[9] = gSegA7
        SegmentRef[10] = gSegA6
        SegmentRef[11] = gSegA5
        SegmentRef[12] = gSegA4
        SegmentRef[13] = gSegA3
        SegmentRef[14] = gSegA2
      Position = Absolute
        SegmentRef = gSegA1
        SegmentCountDirection = RightToLeft
        Translation:
          X = 0.0
          Y = 0.0
          Z = 0.0
        Orientation:
          Angle1 = 0.0
          Angle2 = 0.0
          Angle3 = 0.0
    Track[2]:
      Segments:
        SegmentRef[1] = ::gSegB5
        SegmentRef[2] = ::gSegB4
        SegmentRef[3] = ::gSegB3
        SegmentRef[4] = ::gSegB2
        SegmentRef[5] = ::gSegB1
        SegmentRef[6] = ::gSegB18
        SegmentRef[7] = ::gSegB17
      Position = RelativeToOne
        TrackSegmentPosition:
          SegmentRef = ::gSegB18
        Base:
          SegmentRef = ::gSegA2
          PositionRelativeTo = FromEnd
    Track[3]:
      Segments:
        SegmentRef[1] = ::gSegB15
        SegmentRef[2] = ::gSegB16
      Position = RelativeToOne
        TrackSegmentPosition:
          SegmentRef = ::gSegB16
          PositionRelativeTo = FromEnd
        Base:
          SegmentRef = ::gSegB17
          Position = 0.09
          PositionRelativeTo = FromEnd
    Track[4]:
      Segments:
        SegmentRef[1] = ::gSegB14
        SegmentRef[2] = ::gSegB13
        SegmentRef[3] = ::gSegB12
        SegmentRef[4] = ::gSegB11
        SegmentRef[5] = ::gSegB10
        SegmentRef[6] = ::gSegB9
        SegmentRef[7] = ::gSegB8
      Position = RelativeToOne
        TrackSegmentPosition:
          SegmentRef = ::gSegB14
        Base:
          SegmentRef = ::gSegB15
          Position = 0.09
    Track[5]:
      Segments:
        SegmentRef[1] = ::gSegB6
        SegmentRef[2] = ::gSegB7
      Position = RelativeToOne
        TrackSegmentPosition:
          SegmentRef = ::gSegB6
        Base:
          SegmentRef = ::gSegB5
          Position = 0.09
  CommonSegmentSettings:
    SegmentSimulationOnPLC = On
    CoggingCompensation = Active
      UpperVelLimit = 0.5
    ElongationCompensation = Inactive
    StopReaction = InductionHalt
    SpeedFilter = NotUsed
    ControllerParameters:
      DefaultParameter:
        Controller:
          Position:
            ProportionalGain = 0.0
          Speed:
            ProportionalGain = 0.0
            IntegrationTime = 0.0
          FeedForward:
            TotalMass = 0.0
            ForcePositive = 0.0
            ForceNegative = 0.0
            SpeedForceFactor = 0.0
            ForceLoad = 0.0
        MovementErrorLimits:
          PositionError = 0.004
          VelocityError = 1.2
        Diverter:
          ForceOverride = 1.0
      AdditionalParameterSets = NotUsed
    ScopeOfErrorReaction = Assembly
    ShuttleIdentificationTime = 0
  Shuttles:
    MaxShuttleCount = 50
    MaxShuttleCommandCount = 0
    Deceleration = 0.0
    UseConvoys = Inactive
    DistanceReserve:
      Collision = 0.002
      ErrorStop = 0.006
    ShuttleStereotypes:
      ShuttleStRef[1] = ShuttleStereotype_1
    MagnetPlateConfigurations:
      ShuttleType[1] = 8F1SA.100.xxxxxx-x
    CollisionAvoidance:
      Strategy = Constant
      Exclusion = NotUsed
      MaximumModelDimensions:
        Length:
          ExtentToFront = 0.025
          ExtentToBack = 0.025
        Width:
          Width = 0.046
    Coupling:
      CouplingFeature:
        EliminateShuttleToShuttleDelay = FALSE
  Visualization:
    MonitoringPv
    ProcessingTaskClass = 4
  Alarms = None
```

### Config_3.sector - 5PC900_TS17_00/mappMotion/Config_3.sector
```
Element gSecOvalA (Type=sector)
  Type = Composed
    StartSegment:
      SegmentRef = ::gSegA1
    IntermediateSegments:
      SegmentRef[1] = ::gSegA14
      SegmentRef[2] = ::gSegA13
      SegmentRef[3] = ::gSegA12
      SegmentRef[4] = ::gSegA11
      SegmentRef[5] = ::gSegA10
      SegmentRef[6] = ::gSegA9
      SegmentRef[7] = ::gSegA8
      SegmentRef[8] = ::gSegA7
      SegmentRef[9] = ::gSegA6
      SegmentRef[10] = ::gSegA5
      SegmentRef[11] = ::gSegA4
      SegmentRef[12] = ::gSegA3
    EndSegment:
      SegmentRef = ::gSegA2
      PositionRelativeTo = FromEnd
  Alarms = None
Element gSecOvalB (Type=sector)
  Type = Composed
    StartSegment:
      SegmentRef = ::gSegB1
      PositionRelativeTo = FromEnd
    IntermediateSegments:
      SegmentRef[1] = ::gSegB2
      SegmentRef[2] = ::gSegB3
      SegmentRef[3] = ::gSegB4
      SegmentRef[4] = ::gSegB5
      SegmentRef[5] = ::gSegB6
      SegmentRef[6] = ::gSegB7
      SegmentRef[7] = ::gSegB8
      SegmentRef[8] = ::gSegB9
      SegmentRef[9] = ::gSegB10
      SegmentRef[10] = ::gSegB11
      SegmentRef[11] = ::gSegB12
      SegmentRef[12] = ::gSegB13
      SegmentRef[13] = ::gSegB14
      SegmentRef[14] = ::gSegB15
      SegmentRef[15] = ::gSegB16
      SegmentRef[16] = ::gSegB17
    EndSegment:
      SegmentRef = ::gSegB18
  Alarms = None
Element gSecCompleteLoop (Type=sector)
  Type = Composed
    StartSegment:
      SegmentRef = ::gSegA1
    IntermediateSegments:
      SegmentRef[1] = ::gSegA14
      SegmentRef[2] = ::gSegA13
      SegmentRef[3] = ::gSegA12
      SegmentRef[4] = ::gSegA11
      SegmentRef[5] = ::gSegA10
      SegmentRef[6] = ::gSegA9
      SegmentRef[7] = ::gSegA8
      SegmentRef[8] = ::gSegA7
      SegmentRef[9] = ::gSegA6
      SegmentRef[10] = ::gSegA5
      SegmentRef[11] = ::gSegA4
      SegmentRef[12] = ::gSegA3
      SegmentRef[13] = ::gSegA2
      SegmentRef[14] = ::gSegB1
      SegmentRef[15] = ::gSegB2
      SegmentRef[16] = ::gSegB3
      SegmentRef[17] = ::gSegB4
      SegmentRef[18] = ::gSegB5
      SegmentRef[19] = ::gSegB6
      SegmentRef[20] = ::gSegB7
      SegmentRef[21] = ::gSegB8
      SegmentRef[22] = ::gSegB9
      SegmentRef[23] = ::gSegB10
      SegmentRef[24] = ::gSegB11
      SegmentRef[25] = ::gSegB12
      SegmentRef[26] = ::gSegB13
      SegmentRef[27] = ::gSegB14
      SegmentRef[28] = ::gSegB15
      SegmentRef[29] = ::gSegB16
      SegmentRef[30] = ::gSegB17
    EndSegment:
      SegmentRef = ::gSegB18
  Alarms = MpAlarmX
```

### Config_4.processpointlist - 5PC900_TS17_00/mappMotion/Config_4.processpointlist
```
Element ProcessPointList_1 (Type=processpointlist)
```

### CfgAlList.mpalarmxcore - 5PC900_TS17_00/mappServices/CfgAlList.mpalarmxcore
```
Element gAlarmXCore (Type=mpalarmxcore)
  mapp.AlarmX.Core:
    BySeverity:
      [0]:
        Severity = 10
        [0] = Reaction
          Name = ActWarning
      [1]:
        Severity = 50
        [0] = Reaction
          Name = ActErrorMed
      [2]:
        Severity = 100
        [0] = Reaction
          Name = ActError
    Default:
      [0] = Remain
  mapp.AlarmX.Core.Configuration:
    [0]:
      Name = AL_AlarmMeldung
      Message = AlarmMeldung
      Code = 100
      Severity = 100
      Behavior = DiscreteValueMonitoring
        Monitoring:
          MonitoredPV = ::AlarmXTask:tmpErrorID
          TriggerValues:
            [0] = 100
    [1]:
      Name = AL_AlarmMeldung1
      Message = AlarmMeldung
      Code = 101
      Severity = 100
      Behavior = DiscreteValueMonitoring
        Monitoring:
          MonitoredPV = ::AlarmXTask:tmpErrorID
          TriggerValues:
            [0] = 101
    [2]:
      Name = AL_AlarmMedMeldung
      Message = AlarmMedMeldung
      Code = 50
      Severity = 50
      Behavior = DiscreteValueMonitoring
        Monitoring:
          MonitoredPV = ::AlarmXTask:tmpErrorID
          TriggerValues:
            [0] = 50
    [3]:
      Name = AL_AlarmMedMeldung1
      Message = AlarmMedMeldung1
      Code = 51
      Severity = 50
      Behavior = DiscreteValueMonitoring
        Monitoring:
          MonitoredPV = ::AlarmXTask:tmpErrorID
          TriggerValues:
            [0] = 51
    [4]:
      Name = AL_Warnung
      Message = Warnung
      Code = 10
      Severity = 10
      Behavior = DiscreteValueMonitoring
        Monitoring:
          MonitoredPV = ::AlarmXTask:tmpErrorID
          TriggerValues:
            [0] = 10
    [5]:
      Name = AL_Warnung1
      Message = Warnung1
      Code = 11
      Severity = 10
      Behavior = DiscreteValueMonitoring
        Monitoring:
          MonitoredPV = ::AlarmXTask:tmpErrorID
          TriggerValues:
            [0] = 11
    [6]:
      Name = AL_Error_TD_WebServices
      Message = Error TD_WebServices: {&Snippet_ErrorID_TD_WebServices}
      Code = 102
      Severity = 100
      Behavior = DiscreteValueMonitoring
        Monitoring:
          MonitoredPV = ::AssCtrl:fbWebServices.Error
          TriggerValues:
            [0] = 1
    [7]:
      Name = AL_Error_TD_Recorder
      Message = Error TD_Recorder: {&Snippet_ErrorID_TD_Recorder}
      Code = 103
      Severity = 100
      Behavior = DiscreteValueMonitoring
        Monitoring:
          MonitoredPV = ::AssCtrl:fbRecorder.Error
          TriggerValues:
            [0] = 1
  mapp.AlarmX.Core.Snippets:
    [0]:
      Key = Snippet_ErrorID_TD_WebServices
      Value:
        PV = ::AssCtrl:fbWebServices.ErrorID
    [1]:
      Key = Snippet_ErrorID_TD_Recorder
      Value:
        PV = ::AssCtrl:fbRecorder.ErrorID
  mapp.AlarmX.Core.Categories:
    [0]:
      Name = CatWarning
      SourceProperty:
        Severity = 10
    [1]:
      Name = CatErrorMed
      SourceProperty:
        Severity = 50
    [2]:
      Name = CatError
      SourceProperty:
        Severity = 100
```

## Logical view

Binary libraries used (declarations not repeated): operator, runtime, astime, AsIecCon, standard, AsBrStr, AsZip, FileIO, AsHttp, brsystem, DataObj, sys_lib, ArEventLog, AsArSdm, MpAlarmX 5.21.0, MpBase, McAcpTrak, McBase 5.22.1, McAxis, CoTrace, MpServer 5.21.0, AsMem, AsUSB, TrakLib, TrakDiag 2.01.0

- Project.language (not shown)

### Package Logical/Libraries - Global libraries

### Assembly.typ
```iecst
TYPE
	AssemblyStepEnum :
		(
		ASM_INIT,
		ASM_GET_INFO,
		ASM_W_READY_FOR_POWER_ON,
		ASM_POWER_IS_OFF,
		ASM_W_POWER_ON,
		ASM_ADD_SIM_SHUTTLES,
		ASM_POWER_IS_ON,
		ASM_START_MOVEMENT,
		ASM_W_POWER_OFF,
		ASM_SIMULATE_ERROR,
		ASM_ERR_GET_INFO := 9000,
		ASM_ERR_POWERING_ON,
		ASM_ERR_POWERING_OFF,
		ASM_ERR_START_MOVEMENT,
		ASM_ERR_ADDING_SHUTTLE,
		ASM_ERR_SIMULATE_ERROR,
		ASM_ERR_GENERAL
		);
	AssemblyResetStepEnum :
		(
		ASMR_NO_ERROR,
		ASMR_W_ACKNOWLEDGE,
		ASMR_RESET,
		ASMR_INTERNAL_ERROR
		);
	AssemblyStatusType : 	STRUCT
		Step : AssemblyStepEnum;
		ResetStep : AssemblyResetStepEnum;
		Disabled : BOOL;
		Ready : BOOL;
		Homing : BOOL;
		Stopping : BOOL;
		ErrorStop : BOOL;
		SimulationOnPlcMode : McAcpTrakSimulationOnPlcEnum;
		Info : McAcpTrakAsmInfoType;
	END_STRUCT;
	AssemblyParaType : 	STRUCT
		NumberOfSimulatedShuttles : USINT;
	END_STRUCT;
	AssemblyCmdType : 	STRUCT
		Reset : BOOL;
		PowerOn : BOOL;
		PowerOff : BOOL;
		Start : BOOL;
		SimEncoderError : BOOL;
		SimChannelError : BOOL;
		SimSegmentError : BOOL;
	END_STRUCT;
	AssemblyType : 	STRUCT
		SizeOf : UDINT; (*size of this struct*)
		Status : AssemblyStatusType;
		Para : AssemblyParaType;
		Cmd : AssemblyCmdType;
	END_STRUCT;
END_TYPE
```

### Program Logical/Trak/AssCtrl

#### Variables.var
```iecst
VAR
	fbStartShuttles : TL_StartShuttlesInSector;
	fbLogResetStep : TD_LogWatchSTRING;
	fbLogStep : TD_LogWatchSTRING;
	fbAddSimShuttle : MC_BR_SecAddShuttle_AcpTrak;
	fbPowerOff : MC_BR_AsmPowerOff_AcpTrak;
	fbPowerOn : MC_BR_AsmPowerOn_AcpTrak;
	fbGetInfo : MC_BR_AsmGetInfo_AcpTrak;
	fbReadInfo : MC_BR_AsmReadInfo_AcpTrak;
	fbReadStatus : MC_BR_AsmReadStatus_AcpTrak;
	fbWebServices : TD_WebServices;
	fbRecorder : TD_Recorder;
	step : AssemblyStepEnum;
	fbAsmReset : MC_BR_AsmReset_AcpTrak;
	fbSegCommandError : TD_SegCommandError;
	assemblyCtrl : AssemblyType;
	shuttleData : ARRAY[0..49] OF McAcpTrakShuttleData;
END_VAR
```

#### Cyclic.st
```iecst
PROGRAM _CYCLIC
//test Mapping Visu Buttons
 assemblyCtrl.Cmd.Start := gVisu.Cmd.DiagnosisPlayButton;

	fbLogStep.EventID := TRAK_BASIC_INFO_ID;

	CASE step OF
		ASM_INIT:
		fbGetInfo( Execute := FALSE ); (* reset fb *)
		fbGetInfo( Execute := TRUE );
		fbPowerOn( Execute := FALSE ); (* reset fb *)
		fbPowerOff( Execute := FALSE ); (* reset fb *)
		step := ASM_GET_INFO;

		ASM_GET_INFO:
		fbLogStep.Signal := 'ASM_GET_INFO';
		IF fbGetInfo.Done THEN
			fbGetInfo( Execute := FALSE ); (* reset fb *)
			assemblyCtrl.Status.SimulationOnPlcMode := fbGetInfo.AssemblyInfo.SimulationOnPlcMode;
			step := ASM_W_READY_FOR_POWER_ON;
		ELSIF fbGetInfo.Error THEN
			fbGetInfo( Execute := FALSE ); (* reset fb *)
			step := ASM_ERR_GET_INFO;
			fbLogStep.EventID := TRAK_BASIC_ERROR_ID;
			fbLogStep.Signal := 'ASM_ERR_GET_INFO';
		ELSE (* busy *)
			fbGetInfo();
		END_IF

		ASM_W_READY_FOR_POWER_ON:
		fbLogStep.Signal := 'ASM_W_READY_FOR_POWER_ON';
		IF assemblyCtrl.Status.Info.ReadyForPowerOn THEN
			IF assemblyCtrl.Status.Info.PowerOn THEN
				step := ASM_POWER_IS_ON;
			ELSE
				step := ASM_POWER_IS_OFF;
			END_IF
		END_IF

		ASM_POWER_IS_OFF:
		fbLogStep.Signal := 'ASM_POWER_IS_OFF';
		IF assemblyCtrl.Cmd.PowerOn THEN
			assemblyCtrl.Cmd.PowerOn := FALSE;
			fbPowerOn( Execute := TRUE );
			step := ASM_W_POWER_ON;
		END_IF

		ASM_ADD_SIM_SHUTTLES:
		fbLogStep.Signal := 'ASM_ADD_SIM_SHUTTLES';
		IF fbAddSimShuttle.Done THEN
			fbAddSimShuttle( Execute := FALSE ); (* reset fb *)
			IF assemblyCtrl.Status.Info.ShuttlesCount >= assemblyCtrl.Para.NumberOfSimulatedShuttles OR assemblyCtrl.Para.NumberOfSimulatedShuttles = 0 THEN
				step := ASM_POWER_IS_ON;
			ELSE
				fbAddSimShuttle.Position := fbAddSimShuttle.Position + 0.06;
				fbAddSimShuttle( Execute := TRUE );
			END_IF
		ELSIF fbAddSimShuttle.Error THEN
			fbAddSimShuttle( Execute := FALSE ); (* reset fb *)
			step := ASM_ERR_ADDING_SHUTTLE;
			fbLogStep.EventID := TRAK_BASIC_ERROR_ID;
			fbLogStep.Signal := 'ASM_ERR_ADDING_SHUTTLE';
		ELSE (* busy *)
			fbAddSimShuttle();
		END_IF

		ASM_W_POWER_ON:
		fbLogStep.Signal := 'ASM_W_POWER_ON';
		IF fbPowerOn.Done AND assemblyCtrl.Status.Info.PowerOn THEN
			fbPowerOn( Execute := FALSE );  (* reset fb *)
			IF assemblyCtrl.Status.Info.ShuttlesCount >= assemblyCtrl.Para.NumberOfSimulatedShuttles THEN
				step := ASM_POWER_IS_ON;
			ELSE
				fbAddSimShuttle( Execute := FALSE ); (* reset fb *)
				fbAddSimShuttle( Execute := TRUE );
				step := ASM_ADD_SIM_SHUTTLES;
			END_IF
		ELSIF fbPowerOn.Error THEN
			fbPowerOn( Execute := FALSE );  (* reset fb *)
			step := ASM_ERR_POWERING_ON;
			fbLogStep.EventID := TRAK_BASIC_ERROR_ID;
			fbLogStep.Signal := 'ASM_ERR_POWERING_ON';
		ELSE (* busy *)
			fbPowerOn();
		END_IF

		ASM_POWER_IS_ON:
		fbLogStep.Signal := 'ASM_POWER_IS_ON';
		IF NOT assemblyCtrl.Status.Info.PowerOn THEN
			step := ASM_POWER_IS_OFF;
		ELSIF assemblyCtrl.Cmd.PowerOff THEN
			assemblyCtrl.Cmd.PowerOff := FALSE;
			fbPowerOff( Execute := TRUE );
			step := ASM_W_POWER_OFF;
		ELSIF assemblyCtrl.Cmd.Start THEN
			assemblyCtrl.Cmd.Start := FALSE;
			fbStartShuttles( Execute := FALSE ); (* reset fb *)
			fbStartShuttles( Execute := TRUE ); (* reset fb *)
			step := ASM_START_MOVEMENT;
		ELSIF assemblyCtrl.Cmd.SimSegmentError THEN
			assemblyCtrl.Cmd.SimSegmentError := FALSE;
			fbSegCommandError( Segment := ADR(gSegB7), Type := TD_SEGERRCMD_SEGMENT, Execute := FALSE );
			fbSegCommandError( Execute := TRUE );
			step := ASM_SIMULATE_ERROR;
		ELSIF assemblyCtrl.Cmd.SimChannelError THEN
			assemblyCtrl.Cmd.SimChannelError := FALSE;
			fbSegCommandError( Segment := ADR(gSegB7), Type := TD_SEGERRCMD_CHANNEL, Execute := FALSE );
			fbSegCommandError( Execute := TRUE );
			step := ASM_SIMULATE_ERROR;
		ELSIF assemblyCtrl.Cmd.SimEncoderError THEN
			assemblyCtrl.Cmd.SimEncoderError := FALSE;
			fbSegCommandError( Segment := ADR(gSegB7), Type := TD_SEGERRCMD_ENCODER, Execute := FALSE );
			fbSegCommandError( Execute := TRUE );
			step := ASM_SIMULATE_ERROR;
		END_IF

		ASM_START_MOVEMENT:
		fbLogStep.Signal := 'ASM_START_MOVEMENT';
		IF fbStartShuttles.Done THEN
			fbStartShuttles( Execute := FALSE ); (* reset fb *)
			step := ASM_POWER_IS_ON;
		ELSIF fbStartShuttles.Error THEN
			fbStartShuttles( Execute := FALSE ); (* reset fb *)
			step := ASM_ERR_START_MOVEMENT;
			fbLogStep.EventID := TRAK_BASIC_ERROR_ID;
			fbLogStep.Signal := 'ASM_ERR_START_MOVEMENT';
		ELSE (* busy *)
			fbStartShuttles();
		END_IF

		ASM_SIMULATE_ERROR:
		fbLogStep.Signal := 'ASM_SIMULATE_ERROR';
		IF fbSegCommandError.Done THEN
			fbSegCommandError( Execute := FALSE );
			step := ASM_POWER_IS_ON;
		ELSIF fbSegCommandError.Error THEN
			fbSegCommandError( Execute := FALSE );
			step := ASM_POWER_IS_ON;
//			step := ASM_ERR_SIMULATE_ERROR;
//			fbLogStep.EventID := TRAK_BASIC_ERROR_ID;
//			fbLogStep.Signal := 'ASM_ERR_SIMULATE_ERROR';
		ELSE (* busy *)
			fbSegCommandError();
		END_IF

		ASM_W_POWER_OFF:
		fbLogStep.Signal := 'ASM_W_POWER_OFF';
		IF fbPowerOff.Done OR  NOT assemblyCtrl.Status.Info.PowerOn THEN
			step := ASM_POWER_IS_OFF;
			fbPowerOff( Execute := FALSE ); (* reset fb *)
		ELSIF fbPowerOff.Error THEN
			fbPowerOff( Execute := FALSE ); (* reset fb *)
			step := ASM_ERR_POWERING_OFF;
			fbLogStep.EventID := TRAK_BASIC_ERROR_ID;
			fbLogStep.Signal := 'ASM_ERR_POWERING_OFF';
		ELSE (* busy *)
			fbPowerOff();
		END_IF

		ASM_ERR_GET_INFO..ASM_ERR_GENERAL:

	END_CASE

	assemblyCtrl.Status.Step := step;
	fbLogStep(); (* log steps *)

	fbReadStatus();
	assemblyCtrl.Status.Disabled  	:= fbReadStatus.AssemblyDisabled;
	assemblyCtrl.Status.ErrorStop 	:= fbReadStatus.AssemblyErrorStop;
	assemblyCtrl.Status.Homing 		:= fbReadStatus.AssemblyHoming;
	assemblyCtrl.Status.Stopping 	:= fbReadStatus.AssemblyStopping;
	assemblyCtrl.Status.Ready 	  	:= fbReadStatus.AssemblyReady;

	fbReadInfo();
	assemblyCtrl.Status.Info := fbReadInfo.AssemblyInfo;

	fbRecorder( Trigger := assemblyCtrl.Status.ErrorStop );
	fbWebServices();

	fbLogResetStep.EventID := TRAK_BASIC_INFO_ID;
	CASE assemblyCtrl.Status.ResetStep OF
		ASMR_NO_ERROR:
		fbLogResetStep.Signal := 'ASMR_NO_ERROR';
		IF assemblyCtrl.Status.ErrorStop THEN
			fbAsmReset( Execute := FALSE ); (* reset fb *)
			assemblyCtrl.Cmd.Reset := FALSE;
			assemblyCtrl.Status.ResetStep := ASMR_W_ACKNOWLEDGE;
		END_IF

		ASMR_W_ACKNOWLEDGE:
		fbLogResetStep.Signal := 'ASMR_W_ACKNOWLEDGE';
		IF assemblyCtrl.Cmd.Reset THEN
			assemblyCtrl.Cmd.Reset := FALSE;
			fbAsmReset( Execute := TRUE ); (* reset fb *)
			assemblyCtrl.Status.ResetStep := ASMR_RESET;
		END_IF

		ASMR_RESET:
		fbLogResetStep.Signal := 'ASMR_RESET';
		IF fbAsmReset.Done THEN
			fbAsmReset( Execute := FALSE ); (* reset fb *)
			assemblyCtrl.Status.ResetStep := ASMR_NO_ERROR;
		ELSIF fbAsmReset.Error THEN
			fbAsmReset( Execute := FALSE ); (* reset fb *)
			assemblyCtrl.Status.ResetStep := ASMR_INTERNAL_ERROR;
			fbLogResetStep.EventID := TRAK_BASIC_ERROR_ID;
			fbLogResetStep.Signal := 'ASMR_INERNAL_ERROR';
		ELSE (* busy *)
			fbAsmReset();
		END_IF

		ASMR_INTERNAL_ERROR:

	END_CASE

	fbLogResetStep();

END_PROGRAM
```

#### Init.st
```iecst
PROGRAM _INIT
	gSecOvalA;
	gSecOvalB;
	gSecCompleteLoop;

	fbReadStatus.Assembly := ADR(gAssembly_1);
	fbReadStatus.Enable := TRUE;

	fbReadInfo.Assembly := fbReadStatus.Assembly;
	fbReadInfo.Enable := TRUE;

	fbGetInfo.Assembly := fbReadStatus.Assembly;

	fbPowerOn.Assembly := fbReadStatus.Assembly;

	fbPowerOff.Assembly := fbReadStatus.Assembly;

	fbStartShuttles.Sector := gSecCompleteLoop;
	fbStartShuttles.TargetSector := gSecCompleteLoop;
	fbStartShuttles.Acceleration := 4.0;
	fbStartShuttles.Deceleration := 4.0;
	fbStartShuttles.Velocity := 2.0;
	fbStartShuttles.Jerk := 0.0;
	fbStartShuttles.Direction := mcDIR_POSITIVE;

	fbAddSimShuttle.Sector := ADR(gSecCompleteLoop);
	fbAddSimShuttle.Position := 0.5;

	fbAddSimShuttle.AdvancedParameters.Velocity := 0.0;
	fbAddSimShuttle.AdvancedParameters.Orientation := mcDIR_POSITIVE;
	fbAddSimShuttle.AdvancedParameters.Deceleration := 6.0;
	fbAddSimShuttle.AdvancedParameters.Virtual := FALSE;

	fbAsmReset.Assembly := ADR(gAssembly_1);

	fbRecorder.AssemblyName := 'gAssembly_1';
	fbRecorder.FileDeviceName := 'Diagnosis';
	fbRecorder.DataAddress := ADR(shuttleData);
	fbRecorder.DataSize := SIZEOF(shuttleData); (* type of McAcpTrakShuttleData[] if no shuttle user data is defined, see MC_BR_AsmCopyShuttleData_AcpTrak *)
	fbRecorder.UserDataSize := 0;
	fbRecorder.Enable := TRUE;

	fbWebServices.AssemblyName := fbRecorder.AssemblyName;
	fbWebServices.DataAddress := fbRecorder.DataAddress;
	fbWebServices.DataSize := fbRecorder.DataSize;
	fbWebServices.UserDataSize := fbRecorder.UserDataSize;
	fbWebServices.Enable := TRUE;

	assemblyCtrl.Para.NumberOfSimulatedShuttles := 10;
	assemblyCtrl.SizeOf := SIZEOF(assemblyCtrl);

	step := ASM_INIT;

	fbLogStep( Enable := FALSE, LogName := 'MyTrak', SignalName := 'AssCtrl Step', EventID := TRAK_BASIC_INFO_ID );
	fbLogStep.Enable := TRUE;

	fbLogResetStep( Enable := FALSE, LogName := 'MyTrak', SignalName := 'AssCtrl ResetStep', EventID := TRAK_BASIC_INFO_ID );
	fbLogResetStep.Enable := TRUE;
END_PROGRAM
```

- Visualisation Logical/VisuPackage (not shown)

- Visualisation Logical/mappView (not shown)

### ExplorerVariables.var
```iecst
VAR CONSTANT
	EXPL_DIR_PATH_LENGTH : UINT := 200; (*Maximum length for the complete path *)
	EXPL_LIST_NUM : UINT := 100; (*Maximum number if files and folders that can be listed *)
	EXPL_ITEM_LENGTH : USINT := 50; (*Maximum length for a file or folder name *)
	EXPL_SIZE_LENGTH : USINT := 15; (*Maximum length for a file or folder size*)
	EXPL_UPLOAD_DOWNLOAD_SIZE : UDINT := 5000000; (*Maximum size of memory allocated for uploading and downloading files*)
	EXPL_DEVICE_LIST : ARRAY[0..6] OF STRING[40] := ['USER','SYSTEM','USB_DEVICE1','USB_DEVICE2','USB_DEVICE3','NET_DEVICE','']; (*List of predefined devices *)
END_VAR
VAR
	EXPL_VIEW_FILTER : ARRAY[0..9] OF STRING[5] := ['csv','xml','txt','bmp','jpg',5('')]; (*Files extensions than can be used with the view command*)
	EXPL : expMAIN; (*Explorer main structure*)
END_VAR
```

### Program Logical/mappFileExplorer/FileExplorer (IEC)
